//						mcHeight2MoveAbsolute.Execute		:=	TRUE;
//						mcHeight2MoveAbsolute.Position		:=	lrHeightReadyPosition;
//						IF mcHeight1MoveAbsolute.Done AND mcHeight2MoveAbsolute.Done THEN
//							mcHeight1MoveAbsolute.Execute	:=	FALSE;
//							mcHeight2MoveAbsolute.Execute	:=	FALSE;
//							eState							:=	E_Station.eReady;
//						END_IF	
//					ELSE
							eState							:=	E_Station.eReady;
//					END_IF	
			END_IF

	/////////////////////////////
		E_Station.eHoming:						// Stan bazowania 

			Homing();
			IF NOT bHoming THEN
			  	eState							:=	E_Station.ePreparingToReady;
			   	mcCartesianYManualMove.JogBackwards		:=FALSE;
				mcCartesianZManualMove.JogBackwards		:=FALSE;
				mcPreScrewerManualMove.JogBackwards		:=FALSE;
				mcCatcherManualMove.JogBackwards		:=FALSE;
				
				mcCartesianYManualMove.JogForward		:=FALSE;
				mcCartesianZManualMove.JogForward		:=FALSE;
				mcPreScrewerManualMove.JogForward		:=FALSE;
				mcCatcherManualMove.JogForward			:=FALSE;			
			END_IF		
			
	/////////////////////////////
		E_Station.eHomingDone:                  // Stan wykonania bazowania 
		
			bAdvancedHoming							:= FALSE;
			mcCartesianYManualMove.JogBackwards		:= FALSE;
			mcCartesianZManualMove.JogBackwards		:= FALSE;
			mcPreScrewerManualMove.JogBackwards		:= FALSE;
			mcCatcherManualMove.JogBackwards		:= FALSE;
			                                           
			mcCartesianYManualMove.JogForward		:= FALSE;
			mcCartesianZManualMove.JogForward		:= FALSE;
			mcPreScrewerManualMove.JogForward		:= FALSE;
			mcCatcherManualMove.JogForward			:= FALSE;
			                                           
			bHomingDone								:= TRUE;
			IF NOT bHoming THEN                 	
				eRunningState						:= E_CapPreScrewer.eReady;
			   	eState								:= E_Station.eReady;
			END_IF
			
	/////////////////////////////
		E_Station.ePreparingToReady:            // Stan przygotowywania do gotowosci (zawsze przed Ready)  

		//	IF tonDelayServoOn.Q(*bySafetyStateScrewer1.0 AND bySafetyStateScrewer2.0 AND bySafetyStateHightServo.0 *)THEN
				bCartesianYServoPower	:= nAxisYSafetyState.0;	// Przy pierwszym uruchomieniu Ustawienia Fabryczne robimy na wartość maksymalną
				bCartesianZServoPower	:= nAxisZSafetyState.0;	// Przy pierwszym uruchomieniu Ustawienia Fabryczne robimy na wartość maksymalną
				bPreScrewerPower		:= nAxisScrewSafetyState.0;
				bCatcherPower			:= nAxisCatcherSafetyState.0;
//				bStrawCatcherLiftEnable	:= TRUE;
		//	END_IF	
			
			IF mcCartesianYPower.Status AND mcCartesianZPower.Status AND mcPreScrewerPower.Status AND mcCatcherPower.Status  THEN 

				IF NOT bAxisYInPosition OR NOT bAxisZInPosition OR NOT bCartesianInReadyPos  THEN
					bHomingDone							:= FALSE;
					bHomingWithoutJiesang				:= fbStrawCatcherLift.bHomingDone;
				END_IF	
				 		
				eState									:=	E_Station.eReady;
			END_IF
			
         	IF bIgnoreError THEN
				eState										:=	E_Station.eReady;
			END_IF
	
	/////////////////////////////
		E_Station.ePreparingToDisable:          // Stan przygotowywania do nieaktywnosci (po wyłączeniu Enable) 
  
			bCartesianYServoPower	:= TRUE;	// Przy pierwszym uruchomieniu Ustawienia Fabryczne robimy na wartość maksymalną
			bCartesianZServoPower	:= TRUE;	// Przy pierwszym uruchomieniu Ustawienia Fabryczne robimy na wartość maksymalną
			bPreScrewerPower		:= TRUE;
			bCatcherPower			:= TRUE;
			
			eRunningState					:=	E_CapPreScrewer.eReady;		//Dodane
			PreparingToDisable();

         	IF bIgnoreError THEN
				eState:=E_Station.eDisabled;
			END_IF
			
	/////////////////////////////
		E_Station.eReady:						// Stan gotowosci 
		
		//Detekcja utraconej nasadki
			GVL_UVFF.ftVacuumSensor1(CLK := tonSuckedOk[1].Q);
			GVL_UVFF.ftVacuumSensor2(CLK := tonSuckedOk[2].Q);
			GVL_UVFF.ftVacuumSensor3(CLK := tonSuckedOk[3].Q);
			GVL_UVFF.ftVacuumSensor4(CLK := tonSuckedOk[4].Q);
		
				//Jeżeli utracimy nasadkę--> wyłącz ssawkę
			//bCapSucker[1]					R= GVL.ftVacuumSensor1.Q;
			//bCapSucker[2]					R= GVL.ftVacuumSensor2.Q;
			//bCapSucker[3]					R= GVL.ftVacuumSensor3.Q;
			//bCapSucker[4]					R= GVL.ftVacuumSensor4.Q;
			
			bEnableLift					:= FALSE;
		
		//Zdejmuję HomingDone gdy utracę bodaj jedną nasadkę lub Jiesang nie jest zbazowany
			//IF (*bAnyCapLost OR*) (NOT fbBottleCatch1Station.bHomingDone AND NOT bManualMovement) THEN
			//	bHomingDone					:= FALSE;
			//	bHomingWithoutJiesang		:= fbBottleCatch1Station.bHomingDone;
			//END_IF
		
			(*Skasowanie wszystkich komend*)
			IF rtResetCommands.Q THEN	
				ResetCommands();	
			END_IF
			
			IF bPreRun THEN
				eState						:= E_Station.eStarting;
			END_IF
			
			IF bRun AND NOT bCycleDone (*AND NOT bCycleNotDone*) AND bHomingDone THEN
				eState 						:= E_Station.eRunning; 
			END_IF
			IF bHoming THEN
				eState 						:= E_Station.eHoming; 
			END_IF
			
			IF NOT bRun THEN
				GVL_VIS.bCapSorterPreScrewerBottleCatcherCatch	:= FALSE;
				bPlaceDone										:= FALSE;
				bCycleDone 										:= FALSE;		
			END_IF
			
			IF bManualMovement THEN
				//Jeśli przejście w tryb ruchów manualnych przepisz wszystkie stany siłowników sterowanych przez moduł
				//aby zapobiec ewentualnym kolizjom po wejściu w tryb serwisowy
				//Ruchy manualne siłownika na wózku	
				bManualCapSucker1							:= bCapSucker[1];	
				bmanualCapSucker2							:= bCapSucker[2];	
				bManualCapSucker3							:= bCapSucker[3];	
				bManualCapSucker4							:= bCapSucker[4];	
				                          	    		                 
				bManualCapBlower1							:= bCapBlower1;	
				bManualCapBlower2							:= bCapBlower2;	
				bManualCapBlower3							:= bCapBlower3;	
				bManualCapBlower4							:= bCapBlower4;	
				                          		    	                 
				bManualCapCatcher1							:= bCapCatcher1;
				bManualCapCatcher2							:= bCapCatcher2;
				bManualCapCatcher3							:= bCapCatcher3;
				bManualCapCatcher4					    	:= bCapCatcher4;
				                                        	
				bManualStrawCatchersOpen					:= bStrawCatchersOpen;
				bManualStrawCatchersClose					:= bStrawCatchersClose;	                                            	
				                                        	
			    bManualStrawCatcherActuatorOut 				:= bStrawCatcherActuatorOut;
			    bManualStrawCatcherActuatorIn 				:= bStrawCatcherActuatorIn;
				
				bHomingWithoutJiesang						:= fbStrawCatcherLift.bHomingDone;
				
				eState 										:=	E_Station.eManualMovement; 

			END_IF
			
	/////////////////////////////
		E_Station.eStopping:					// Stan zatrzymywania 
			
			RunningCam();//RunningWithFlyingSaw();				//Running();
			
					IF bStopAllowed THEN
						eState 								:=	E_Station.eReady;
					END_IF

				
	/////////////////////////////
		E_Station.eStarting:                  	// Stan uruchamiania (po Ready)				
		
		IF 	eRunningState = E_CapPreScrewer.eReady THEN	//Jeżeli jesteśmy na poz. ready--> sprawdź i dojedź do pozycji home
				//Dojazd do poz top		                                                    	
			mcCartesianZMoveAbsolute.Execute						:= NOT bAxisZInTopPos;		
			mcCartesianZMoveAbsolute.Position						:= stParameters.lrTopZPosition;
			mcCartesianZMoveAbsolute.Acceleration					:= 500.0;
			mcCartesianZMoveAbsolute.Deceleration					:= 500.0;
			mcCartesianZMoveAbsolute.Velocity						:= 50;
			                                        				
			//najpierw os Z potem winda chwytakow   				
			mcCatcherMoveAbsolute.Execute							:= NOT bAxisStrawCatcherHomePos AND bAxisZInTopPos;		
			mcCatcherMoveAbsolute.Position							:= stParameters.lrCatcherCatchingPosition;
			mcCatcherMoveAbsolute.Acceleration						:= 300.0;
			mcCatcherMoveAbsolute.Deceleration						:= 300.0;
			mcCatcherMoveAbsolute.Velocity							:= 30;
			                                        				
			mcCartesianYMoveAbsolute.Execute						:= NOT bAxisYInHomePos AND bAxisZInTopPos;
			mcCartesianYMoveAbsolute.Position						:= stParameters.lrPickYPosition;
			mcCartesianYMoveAbsolute.Acceleration					:= 500.0;
			mcCartesianYMoveAbsolute.Deceleration					:= 500.0;
			mcCartesianYMoveAbsolute.Velocity						:= 50; 
			                                                    	
			IF bAxisZInTopPos THEN
				GVL_VIS.bCapSorterPreScrewerCatchStationHoming			:= NOT fbStrawCatcherLift.bHomingDone;
				GVL_VIS.bCapSorterPreScrewerCatcherStationHeightSet		:= NOT GVL_VIS.bCapSorterPreScrewerCatchStationHoming AND NOT bStrawCatcherLiftInHomePos;
				bEnableLift												:= TRUE;
			END_IF
    		
				IF 	bCartesianInTopPos AND bStrawCatcherLiftInHomePos THEN
					mcCartesianZMoveAbsolute.Execute              	:= FALSE;
					mcCatcherMoveAbsolute.Execute                 	:= FALSE;
					mcCartesianYMoveAbsolute.Execute              	:= FALSE;
					GVL_VIS.bCapSorterPreScrewerCatchStationHoming	:= FALSE;
					eState											:= E_Station.eRunning; 
				END_IF
		ELSE
			eState							:= E_Station.eRunning; 
			bEnableLift						:= TRUE;	
		END_IF	
					
			
	/////////////////////////////
		E_Station.eRunning:               		// Stan wykonywania cyklu (po Startingu), w tym stanie osobny
		
 			IF bRun THEN
				IF bSimulationEna THEN
					Simulation();
				ELSE	
					RunningCam();	//RunningWithFlyingSaw();				//Running();
				END_IF
				
				
			ELSIF NOT bPreRun THEN
				bBottleCatcherCatchTemp		:= FALSE;
				eState 				 		:= E_Station.eStopping;		
			END_IF
				
			
	/////////////////////////////	
		E_Station.eDone:
		
			IF bCycleDone THEN (*Cykl zakończony*)
				bBottleCatcherCatchTemp		:= FALSE;
			END_IF	
			
			IF NOT bPreRun  AND bStopAllowed THEN					(*Przerywanie cyklu*)
				bBottleCatcherCatchTemp		:= FALSE;
				eState 				 		:= E_Station.eStopping;	
			ELSIF NOT bRun THEN
				GVL_VIS.bCapSorterPreScrewerBottleCatcherCatch	:= FALSE;
				bPlaceDone										:= FALSE;
				bCycleDone 										:= FALSE;	
				eState 				 							:= E_Station.eRunning;	
			END_IF
		
		
		
	END_CASE

	
//IF (ABS(GVL_VIS.lrCapSorterPreScrewerCatcherStationHeightCV-stParameters.lrCatcherHightSV) > 2) AND
//	(eState = E_Station.eStarting OR eState = E_Station.ePreparingToReady) THEN
//			GVL_VIS.bCapSorterPreScrewerCatcherStationHeightSet 				:= TRUE;
//ELSIF ABS(GVL_VIS.lrCapSorterPreScrewerCatcherStationHeightCV-stParameters.lrCatcherHightSV) < 2 THEN
//			GVL_VIS.bCapSorterPreScrewerCatcherStationHeightSet 				:= FALSE;	
//END_IF
END_ACTION

ACTION ErrorHandling:
//CZYTANIE STATUSÓW
CartesianYAxisRef.ReadStatus();
CartesianZAxisRef.ReadStatus();
CatcherAxisRef.ReadStatus();
PreScrewerAxisRef.ReadStatus();
//Czasówki od siłowników
tonErrorStrawCatcherIn(IN:= bStrawCatcherActuatorIn AND NOT bStrawCatcherIn,PT:=T#1000MS);
tonErrorStrawCatcherOut(IN:= bStrawCatcherActuatorOut AND NOT bStrawCatcherOut,PT:=T#1000MS);



//**********************LISTA BŁĘDÓW******************************
bStateError	:= (eState=E_Station.eError) OR (eState=E_Station.eResetting) OR NOT bEstop OR bIgnoreError;

//PreparingToDisable i StateError ze względu na wciśnięcie EStopa podczas wyłączania i pojawienie się blędu
IF bEnable OR eState=E_Station.ePreparingToDisable THEN
	


	//Error 1 - BŁĄD SERWA POZIOMEGO X
	IF (CartesianYAxisRef.Status.Error OR mcCartesianYMoveAbsolute.Error) AND NOT arrFbAllarm[0].bActive THEN
		sAxisAlarm := CONCAT(UDINT_TO_STRING(CartesianYAxisRef.Status.ErrorID),F_AxErrMsg(CartesianYAxisRef.Status.ErrorID));
		arrFbAllarm[0].ipArguments.Clear().AddString(sAxisAlarm);		
		arrFbAllarm[0].Raise(nTimeStamp := 0);		
		udiErrorID							:=	1129;
		udiCartesianXServoErrorNr			:=	CartesianYAxisRef.Status.ErrorID;
		sErrorDescription					:=	'Błąd napędu poziomego Y. Błąd NC:';
		sErrorDescription2					:=	F_AX8xErrMsg(TO_UINT(udiCartesianXServoErrorNr));
	ELSIF NOT CartesianYAxisRef.Status.Error AND NOT mcCartesianYMoveAbsolute.Error AND eState = E_Station.eResetting AND arrFbAllarm[0].bActive THEN
			arrFbAllarm[0].Clear(nTimeStamp := 0, bResetConfirmation := FALSE);
	END_IF;
	
	//Error 2 - BŁĄD SERWA PIONOWEGO Z
	IF (CartesianZAxisRef.Status.Error OR mcCartesianZMoveAbsolute.Error) AND NOT arrFbAllarm[1].bActive THEN
		sAxisAlarm := CONCAT(UDINT_TO_STRING(CartesianZAxisRef.Status.ErrorID),F_AxErrMsg(CartesianZAxisRef.Status.ErrorID));
		arrFbAllarm[1].ipArguments.Clear().AddString(sAxisAlarm);		
		arrFbAllarm[1].Raise(nTimeStamp := 0);		
		udiErrorID							:=	1130;
		udiCartesianZServoErrorNr			:=	CartesianZAxisRef.Status.ErrorID;
		sErrorDescription					:=	'Błąd napędu podnoszenia Z. Błąd NC:';
		sErrorDescription2					:=	F_AX8xErrMsg(TO_UINT(udiCartesianZServoErrorNr));
	ELSIF NOT CartesianZAxisRef.Status.Error AND NOT mcCartesianZMoveAbsolute.Error AND eState = E_Station.eResetting AND arrFbAllarm[1].bActive THEN
			arrFbAllarm[1].Clear(nTimeStamp := 0, bResetConfirmation := FALSE);
	END_IF;
	
	//Error 3 - BŁĄD SERWA PIONOWEGO UCHWYTU SŁOMEK
	IF (CatcherAxisRef.Status.Error OR mcCatcherMoveAbsolute.Error) AND NOT arrFbAllarm[2].bActive THEN		
		sAxisAlarm := CONCAT(UDINT_TO_STRING(CatcherAxisRef.Status.ErrorID),F_AxErrMsg(CatcherAxisRef.Status.ErrorID));
		arrFbAllarm[2].ipArguments.Clear().AddString(sAxisAlarm);		
		arrFbAllarm[2].Raise(nTimeStamp := 0);		
		udiErrorID							:=	1131;
		udiCatcherServoErrorNr				:=	CatcherAxisRef.Status.ErrorID;
		sErrorDescription					:=	'Błąd napędu podnoszenia chwytaka słomek. Błąd NC:';
		sErrorDescription2					:=	F_AX8xErrMsg(TO_UINT(udiCatcherServoErrorNr));
	ELSIF NOT CatcherAxisRef.Status.Error AND NOT  mcCatcherMoveAbsolute.Error AND eState = E_Station.eResetting AND arrFbAllarm[2].bActive THEN
			arrFbAllarm[2].Clear(nTimeStamp := 0, bResetConfirmation := FALSE);
	END_IF;
	
	//Error 4 - BŁĄD SERWA OBROTOWEGO
	IF (PreScrewerAxisRef.Status.Error OR mcPreScrewerMoveAbsolute.Error OR bTestError) AND NOT arrFbAllarm[3].bActive THEN
		sAxisAlarm := CONCAT(UDINT_TO_STRING(PreScrewerAxisRef.Status.ErrorID),F_AxErrMsg(PreScrewerAxisRef.Status.ErrorID));
		arrFbAllarm[3].ipArguments.Clear().AddString(sAxisAlarm);		
		arrFbAllarm[3].Raise(nTimeStamp := 0);		
		udiErrorID							:=	1132;
		udiPreScrewerServoErrorNr			:=	PreScrewerAxisRef.Status.ErrorID;
		sErrorDescription					:=	'Błąd napędu zakręcania. Błąd NC:';
		sErrorDescription2					:=	F_AX8xErrMsg(TO_UINT(udiPreScrewerServoErrorNr));
	ELSIF NOT PreScrewerAxisRef.Status.Error AND NOT  mcPreScrewerMoveAbsolute.Error AND eState = E_Station.eResetting AND arrFbAllarm[3].bActive THEN
			arrFbAllarm[3].Clear(nTimeStamp := 0, bResetConfirmation := FALSE);
	END_IF;
	
	IF PreScrewerAxisRef.Status.Error THEN
		GVL_UVFF.diTest1	:= GVL_UVFF.diTest1 + 1;
	END_IF
	
	IF mcPreScrewerMoveAbsolute.Error THEN
		GVL_UVFF.diTest2	:= GVL_UVFF.diTest2 + 1;
	END_IF
	
	IF mcPreScrewerMoveRelative.Error THEN
		GVL_UVFF.diTesy3	:= GVL_UVFF.diTesy3 + 1;
	END_IF
	
	IF bTestError THEN
		GVL_UVFF.diTest4	:= GVL_UVFF.diTest4 + 1;
	END_IF	
	
	
	
	
	
	//Error 5A - BŁĄD PRZEKROCZENIE CZASU DZIAŁANIA SIŁOWNIKA CHWYTAKÓW SŁOMEK
	IF tonErrorStrawCatcherOut.Q AND NOT arrFbAllarm[4].bActive THEN
		arrFbAllarm[4].Raise(nTimeStamp := 0);	
		udiErrorID							:=	1133;
		udiPreScrewerServoErrorNr			:=	PreScrewerAxisRef.Status.ErrorID;
		sErrorDescription					:=	'Błąd siłownika chwytaków słomek | Zablokowany wysów';
		sErrorDescription2					:=	'';
	ELSIF NOT tonErrorStrawCatcherOut.Q AND eState = E_Station.eResetting AND arrFbAllarm[4].bActive THEN
			arrFbAllarm[4].Clear(nTimeStamp := 0, bResetConfirmation := FALSE);
	END_IF;
	
	//Error 5B - BŁĄD PRZEKROCZENIE CZASU DZIAŁANIA SIŁOWNIKA CHWYTAKÓW SŁOMEK
	IF tonErrorStrawCatcherIn.Q AND NOT arrFbAllarm[5].bActive THEN
		arrFbAllarm[5].Raise(nTimeStamp := 0);	
		udiErrorID							:=	1134;
		udiPreScrewerServoErrorNr			:=	PreScrewerAxisRef.Status.ErrorID;
		sErrorDescription					:=	'Błąd siłownika chwytaków słomek | Zablokowane cofnięcie';
		sErrorDescription2					:=	'';
	ELSIF NOT tonErrorStrawCatcherIn.Q AND eState = E_Station.eResetting AND arrFbAllarm[5].bActive THEN
			arrFbAllarm[5].Clear(nTimeStamp := 0, bResetConfirmation := FALSE);
	END_IF;
	
	//Error 6 - Blad podnosnika Jiecang - brak zasilania lub zablokowany mechanicznie
	IF fbStrawCatcherLift.bError AND fbStrawCatcherLift.nErrorNr = 1 AND NOT arrFbAllarm[6].bActive THEN
		arrFbAllarm[6].Raise(nTimeStamp := 0);	
    	udiErrorID				:= 1135;
    	sErrorDescription		:= 'Błąd podnosnika lub brak zasilania';
    	sErrorDescription2		:= ' ';
	ELSIF NOT fbStrawCatcherLift.bError AND eState = E_Station.eResetting AND arrFbAllarm[6].bActive THEN
			arrFbAllarm[6].Clear(nTimeStamp := 0, bResetConfirmation := FALSE);
	END_IF;
		

	//Error 6 - Blad podnosnika Jiecang - prak zasilania lub zablokowany mechanicznie
	IF fbStrawCatcherLift.bError AND fbStrawCatcherLift.nErrorNr = 2 AND NOT arrFbAllarm[7].bActive THEN
		arrFbAllarm[7].Raise(nTimeStamp := 0);
    	udiErrorID				:= 1136;
    	sErrorDescription		:= 'Błąd podnosnika  - wartość zadana jest większa od wartości maksymalnej';
    	sErrorDescription2		:= ' ';
	ELSIF NOT fbStrawCatcherLift.bError AND eState = E_Station.eResetting AND arrFbAllarm[7].bActive THEN
			arrFbAllarm[7].Clear(nTimeStamp := 0, bResetConfirmation := FALSE);
	END_IF;
	
	
	//Error 6 - Blad podnosnika Jiecang - prak zasilania lub zablokowany mechanicznie
	IF  fbStrawCatcherLift.bError AND fbStrawCatcherLift.nErrorNr = 3 AND NOT arrFbAllarm[8].bActive THEN
		arrFbAllarm[8].Raise(nTimeStamp := 0);
    	udiErrorID				:= 1137;
    	sErrorDescription		:= 'Błąd podnosnika - wartość zadana jest mniejsza od wartości minimalnej';
    	sErrorDescription2		:= ' ';
	ELSIF NOT fbStrawCatcherLift.bError AND eState = E_Station.eResetting AND arrFbAllarm[8].bActive THEN
			arrFbAllarm[8].Clear(nTimeStamp := 0, bResetConfirmation := FALSE);
	END_IF;
	
		//Error 11 - Blad Kolizja	
	IF  rtCollisionError.Q AND NOT arrFbAllarm[13].bActive THEN
		arrFbAllarm[13].Raise(nTimeStamp := 0);
    	udiErrorID				:= 1142;
    	sErrorDescription		:= 'Kolizja kartezjana z transporterem nakrętek | Zbazuj stacje wkładania nakrętek';
    	sErrorDescription2		:= '';
	ELSIF NOT  rtCollisionError.Q AND eState = E_Station.eResetting AND arrFbAllarm[13].bActive THEN
			arrFbAllarm[13].Clear(nTimeStamp := 0, bResetConfirmation := FALSE);
	END_IF;

		//Przekroczona ilość prób pobrania nasadki, mówer1, słot1
	IF diMover1VacuumRetry[1] >= 3  AND NOT arrFbAllarm[14].bActive THEN
		arrFbAllarm[14].Raise(nTimeStamp := 0);
    	udiErrorID				:= 1143;
    	sErrorDescription		:= 'Przekroczona ilość prób pobrania nasadki, wózek1, slot1';
    	sErrorDescription2		:= '';
	ELSIF diMover1VacuumRetry[1] < 3 AND eState = E_Station.eResetting AND arrFbAllarm[14].bActive THEN
			arrFbAllarm[14].Clear(nTimeStamp := 0, bResetConfirmation := FALSE);
	END_IF;
	
	IF diMover1VacuumRetry[2] >= 3  AND NOT arrFbAllarm[15].bActive THEN
		arrFbAllarm[15].Raise(nTimeStamp := 0);
    	udiErrorID				:= 1144;
    	sErrorDescription		:= 'Przekroczona ilość prób pobrania nasadki, wózek1, slot2';
    	sErrorDescription2		:= '';
	ELSIF diMover1VacuumRetry[2] < 3 AND eState = E_Station.eResetting AND arrFbAllarm[15].bActive THEN
			arrFbAllarm[15].Clear(nTimeStamp := 0, bResetConfirmation := FALSE);
	END_IF;

	IF diMover1VacuumRetry[3] >= 3  AND NOT arrFbAllarm[16].bActive THEN
		arrFbAllarm[16].Raise(nTimeStamp := 0);
    	udiErrorID				:= 1145;
    	sErrorDescription		:= 'Przekroczona ilość prób pobrania nasadki, wózek1, slot3';
    	sErrorDescription2		:= '';
	ELSIF diMover1VacuumRetry[3] < 3 AND eState = E_Station.eResetting AND arrFbAllarm[16].bActive THEN
			arrFbAllarm[16].Clear(nTimeStamp := 0, bResetConfirmation := FALSE);
	END_IF;
	
	IF diMover1VacuumRetry[4] >= 3  AND NOT arrFbAllarm[17].bActive THEN
		arrFbAllarm[17].Raise(nTimeStamp := 0);
    	udiErrorID				:= 1146;
    	sErrorDescription		:= 'Przekroczona ilość prób pobrania nasadki, wózek1, slot4';
    	sErrorDescription2		:= '';
	ELSIF diMover1VacuumRetry[4] < 3 AND eState = E_Station.eResetting AND arrFbAllarm[17].bActive THEN
			arrFbAllarm[17].Clear(nTimeStamp := 0, bResetConfirmation := FALSE);
	END_IF;
	
			//Przekroczona ilość prób pobrania nasadki, mówer2, słot1
	IF diMover2VacuumRetry[1] >= 3  AND NOT arrFbAllarm[18].bActive THEN
		arrFbAllarm[18].Raise(nTimeStamp := 0);
    	udiErrorID				:= 1147;
    	sErrorDescription		:= 'Przekroczona ilość prób pobrania nasadki, wózek2, slot1';
    	sErrorDescription2		:= '';
	ELSIF diMover2VacuumRetry[1] < 3 AND eState = E_Station.eResetting AND arrFbAllarm[18].bActive THEN
			arrFbAllarm[18].Clear(nTimeStamp := 0, bResetConfirmation := FALSE);
	END_IF;
	
	IF diMover2VacuumRetry[2] >= 3  AND NOT arrFbAllarm[19].bActive THEN
		arrFbAllarm[19].Raise(nTimeStamp := 0);
    	udiErrorID				:= 1148;
    	sErrorDescription		:= 'Przekroczona ilość prób pobrania nasadki, wózek2, slot2';
    	sErrorDescription2		:= '';
	ELSIF diMover2VacuumRetry[2] < 3 AND eState = E_Station.eResetting AND arrFbAllarm[19].bActive THEN
			arrFbAllarm[19].Clear(nTimeStamp := 0, bResetConfirmation := FALSE);
	END_IF;

	IF diMover2VacuumRetry[3] >= 3  AND NOT arrFbAllarm[20].bActive THEN
		arrFbAllarm[20].Raise(nTimeStamp := 0);
    	udiErrorID				:= 1149;
    	sErrorDescription		:= 'Przekroczona ilość prób pobrania nasadki, wózek2, slot3';
    	sErrorDescription2		:= '';
	ELSIF diMover2VacuumRetry[3] < 3 AND eState = E_Station.eResetting AND arrFbAllarm[20].bActive THEN
			arrFbAllarm[20].Clear(nTimeStamp := 0, bResetConfirmation := FALSE);
	END_IF;
	
	IF diMover2VacuumRetry[4] >= 3  AND NOT arrFbAllarm[21].bActive THEN
		arrFbAllarm[21].Raise(nTimeStamp := 0);
    	udiErrorID				:= 1150;
    	sErrorDescription		:= 'Przekroczona ilość prób pobrania nasadki, wózek2, slot4';
    	sErrorDescription2		:= '';
	ELSIF diMover2VacuumRetry[4] < 3 AND eState = E_Station.eResetting AND arrFbAllarm[21].bActive THEN
			arrFbAllarm[21].Clear(nTimeStamp := 0, bResetConfirmation := FALSE);
	END_IF;

	IF NOT arrFbAllarm[22].bActive AND (fbVirtualAxis.bErrorFB  OR fbVirtualAxis.bError) THEN	
		sAxisAlarm := CONCAT(UDINT_TO_STRING(fbVirtualAxis.nErrorId),F_AxErrMsg(fbVirtualAxis.nErrorId));
		arrFbAllarm[22].ipArguments.Clear().AddString(sAxisAlarm);		
		arrFbAllarm[22].Raise(nTimeStamp := 0);	
		udiErrorID							:=	1151;
		sErrorDescription					:=	'Błąd wirtualnej osi:';
		sErrorDescription2					:=	F_AX8xErrMsg(TO_UINT(fbVirtualAxis.nErrorId));
	ELSIF NOT fbVirtualAxis.bError AND NOT  fbVirtualAxis.bErrorFB AND eState = E_Station.eResetting AND arrFbAllarm[22].bActive THEN
			arrFbAllarm[22].Clear(nTimeStamp := 0, bResetConfirmation := FALSE);
	END_IF;
	
	IF (fbVirtualAxis.pSetPos.Error OR fbVirtualAxis.pSetPos.CommandAborted) AND NOT arrFbAllarm[23].bActive THEN
		arrFbAllarm[23].ipArguments.Clear().AddUDInt(fbVirtualAxis.pSetPos.ErrorID);		
		arrFbAllarm[23].Raise(nTimeStamp := 0);		
    	udiErrorID							:= 1152;
    	udiErrorID							:= udiErrorID + iStationIndex;
    	sErrorDescription					:= CONCAT('Błąd wirtualnej osi', UDINT_TO_STRING(fbVirtualAxis.pSetPos.ErrorID));
    	sErrorDescription2					:= ' ';	
	ELSIF NOT fbVirtualAxis.pSetPos.Error AND eState = E_Station.eResetting AND arrFbAllarm[23].bActive THEN
			arrFbAllarm[23].Clear(nTimeStamp := 0, bResetConfirmation := FALSE);
	END_IF;
	
	IF fbCamTableSelectAxisZ.Error AND NOT arrFbAllarm[24].bActive THEN
		arrFbAllarm[24].ipArguments.Clear().AddUDInt(fbCamTableSelectAxisZ.ErrorID);		
		arrFbAllarm[24].Raise(nTimeStamp := 0);		
    	udiErrorID							:= 1154;
    	udiErrorID							:= udiErrorID + iStationIndex;
    	sErrorDescription					:= CONCAT('Błąd generowania krzywki osi Z, MC_CamTableSelect.ErrorID:', UDINT_TO_STRING(fbCamTableSelectAxisZ.ErrorID));
    	sErrorDescription2					:= ' ';	
	ELSIF NOT fbCamTableSelectAxisZ.Error AND eState = E_Station.eResetting AND arrFbAllarm[24].bActive THEN
			arrFbAllarm[24].Clear(nTimeStamp := 0, bResetConfirmation := FALSE);
	END_IF;
	
	IF fbCamTableSelectCatcher.Error AND NOT arrFbAllarm[25].bActive THEN
		arrFbAllarm[25].ipArguments.Clear().AddUDInt(fbCamTableSelectCatcher.ErrorID);		
		arrFbAllarm[25].Raise(nTimeStamp := 0);		
    	udiErrorID							:= 1155;
    	udiErrorID							:= udiErrorID + iStationIndex;
    	sErrorDescription					:= CONCAT('Błąd generowania krzywki osi prowadzenia słomki, MC_CamTableSelect.ErrorID:', UDINT_TO_STRING(fbCamTableSelectCatcher.ErrorID));
    	sErrorDescription2					:= ' ';	
	ELSIF NOT fbCamTableSelectCatcher.Error AND eState = E_Station.eResetting AND arrFbAllarm[25].bActive THEN
			arrFbAllarm[25].Clear(nTimeStamp := 0, bResetConfirmation := FALSE);
	END_IF;
	
	IF fbCamInAxisZ.Error AND NOT arrFbAllarm[26].bActive THEN
		arrFbAllarm[26].ipArguments.Clear().AddUDInt(fbCamInAxisZ.ErrorID);		
		arrFbAllarm[26].Raise(nTimeStamp := 0);		
    	udiErrorID							:= 1156;
    	udiErrorID							:= udiErrorID + iStationIndex;
    	sErrorDescription					:= CONCAT('Błąd synchronizacji osi Z, MC_CamIn.ErrorID: ', UDINT_TO_STRING(fbCamInAxisZ.ErrorID));
    	sErrorDescription2					:= ' ';	
	ELSIF NOT fbCamInAxisZ.Error AND eState = E_Station.eResetting AND arrFbAllarm[26].bActive THEN
			arrFbAllarm[26].Clear(nTimeStamp := 0, bResetConfirmation := FALSE);
	END_IF;
	
	IF fbCamInAxisCatcher.Error AND NOT arrFbAllarm[27].bActive THEN
		arrFbAllarm[27].ipArguments.Clear().AddUDInt(fbCamInAxisCatcher.ErrorID);		
		arrFbAllarm[27].Raise(nTimeStamp := 0);		
    	udiErrorID							:= 1157;
    	udiErrorID							:= udiErrorID + iStationIndex;
    	sErrorDescription					:= CONCAT('Błąd synchronizacji osi prowadzenia słomki, MC_CamIn.ErrorID:', UDINT_TO_STRING(fbCamInAxisCatcher.ErrorID));
    	sErrorDescription2					:= ' ';	
	ELSIF NOT fbCamInAxisCatcher.Error AND eState = E_Station.eResetting AND arrFbAllarm[27].bActive THEN
			arrFbAllarm[27].Clear(nTimeStamp := 0, bResetConfirmation := FALSE);
	END_IF;
	
	IF fbCamOutAxisZ.Error AND NOT arrFbAllarm[28].bActive THEN
		arrFbAllarm[28].ipArguments.Clear().AddUDInt(fbCamOutAxisZ.ErrorID);		
		arrFbAllarm[28].Raise(nTimeStamp := 0);		
    	udiErrorID							:= 1158;
    	udiErrorID							:= udiErrorID + iStationIndex;
    	sErrorDescription					:= CONCAT('Błąd rozsynchronizacji osi Z, MCCamOut.ErrorID:', UDINT_TO_STRING(fbCamOutAxisZ.ErrorID));
    	sErrorDescription2					:= ' ';	
	ELSIF NOT fbCamOutAxisZ.Error AND eState = E_Station.eResetting AND arrFbAllarm[28].bActive THEN
			arrFbAllarm[28].Clear(nTimeStamp := 0, bResetConfirmation := FALSE);
	END_IF;
	
	IF fbCamOutAxisCatcher.Error AND NOT arrFbAllarm[29].bActive THEN
		arrFbAllarm[29].ipArguments.Clear().AddUDInt(fbCamOutAxisCatcher.ErrorID);		
		arrFbAllarm[29].Raise(nTimeStamp := 0);		
    	udiErrorID							:= 1159;
    	udiErrorID							:= udiErrorID + iStationIndex;
    	sErrorDescription					:= CONCAT('Błąd rozsynchronizacji osi prowadzenia słomki, MCCamOut.ErrorID:', UDINT_TO_STRING(fbCamOutAxisCatcher.ErrorID));
    	sErrorDescription2					:= ' ';	
	ELSIF NOT fbCamOutAxisCatcher.Error AND eState = E_Station.eResetting AND arrFbAllarm[29].bActive THEN
			arrFbAllarm[29].Clear(nTimeStamp := 0, bResetConfirmation := FALSE);
	END_IF;
	
	FOR i:= 0 TO 23 DO
		bError S= arrFbAllarm[i].bActive;
	END_FOR
	
ELSE
	bError := FALSE;
END_IF


//******************PRZEJŚCIE DO eERROR*****************************


IF bError AND NOT bStateError THEN
	IF eLastState = E_Station.eRunning THEN
		bCycleNotDone 			:= FALSE;
	END_IF
	eState := E_Station.eError;
	ResetCommands();
END_IF

//****************WYŚWIETLANIE STATUSU BLEDU***********************

(*Wyświetlanie błedu na wyjściu*)
bError;

(*Przepisywanie nazwy stacji*)
sErrorStationName := wsLiteral_TO_UTF8(wsStationName);

(*Kasowanie casów resettingu*)
//IF  udiErrorID-iStationIndex <>3 THEN
//	iErrorResseting3	:=	0;
//END_IF
END_ACTION

ACTION FBs:
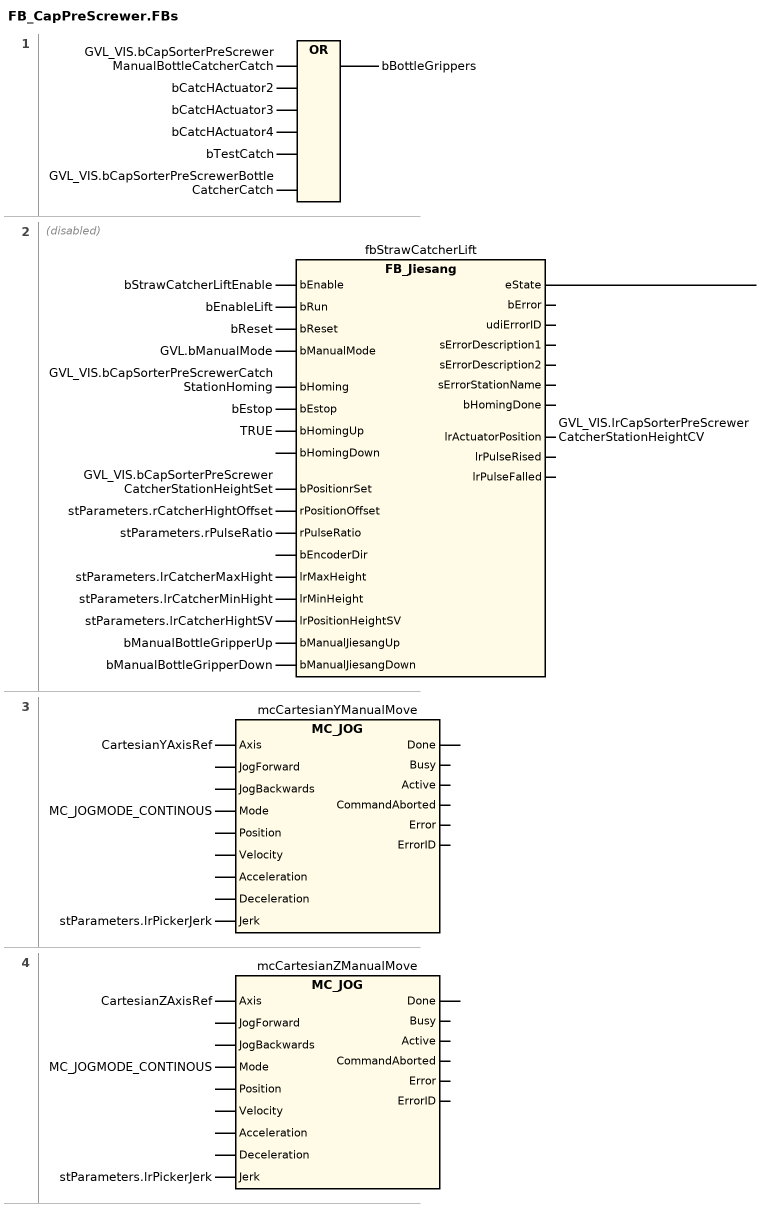
// NETWORK 1
bBottleGrippers := GVL_VIS.bCapSorterPreScrewerManualBottleCatcherCatch OR bCatcHActuator2 OR bCatcHActuator3 OR bCatcHActuator4 OR bTestCatch OR GVL_VIS.bCapSorterPreScrewerBottleCatcherCatch;

// NETWORK 2 (disabled)
// fbStrawCatcherLift(
//     bEnable := bStrawCatcherLiftEnable,
//     bRun := bEnableLift,
//     bReset := bReset,
//     bManualMode := GVL.bManualMode,
//     bHoming := GVL_VIS.bCapSorterPreScrewerCatchStationHoming,
//     bEstop := bEstop,
//     bHomingUp := TRUE,
//     bPositionrSet := GVL_VIS.bCapSorterPreScrewerCatcherStationHeightSet,
//     rPositionOffset := stParameters.rCatcherHightOffset,
//     rPulseRatio := stParameters.rPulseRatio,
//     lrMaxHeight := stParameters.lrCatcherMaxHight,
//     lrMinHeight := stParameters.lrCatcherMinHight,
//     lrPositionHeightSV := stParameters.lrCatcherHightSV,
//     bManualJiesangUp := bManualBottleGripperUp,
//     bManualJiesangDown := bManualBottleGripperDown,
//     lrActuatorPosition => GVL_VIS.lrCapSorterPreScrewerCatcherStationHeightCV); // FB_Jiesang

// NETWORK 3
mcCartesianYManualMove(
    Axis := CartesianYAxisRef,
    Mode := MC_JOGMODE_CONTINOUS,
    Jerk := stParameters.lrPickerJerk); // MC_JOG

// NETWORK 4
mcCartesianZManualMove(
    Axis := CartesianZAxisRef,
    Mode := MC_JOGMODE_CONTINOUS,
    Jerk := stParameters.lrPickerJerk); // MC_JOG

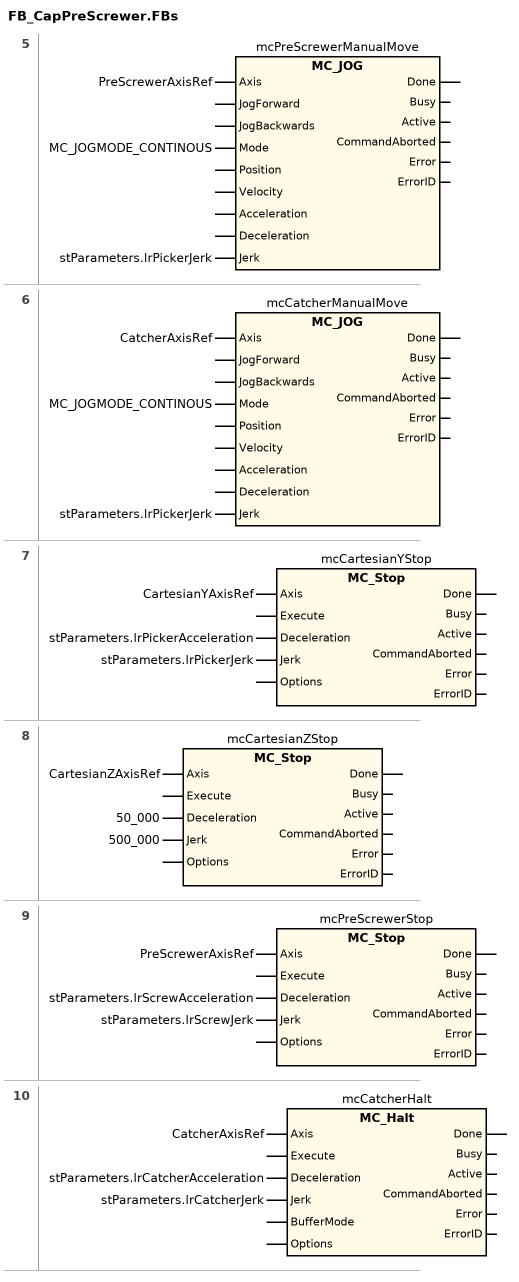
// NETWORK 5
mcPreScrewerManualMove(
    Axis := PreScrewerAxisRef,
    Mode := MC_JOGMODE_CONTINOUS,
    Jerk := stParameters.lrPickerJerk); // MC_JOG

// NETWORK 6
mcCatcherManualMove(Axis := CatcherAxisRef, Mode := MC_JOGMODE_CONTINOUS, Jerk := stParameters.lrPickerJerk); // MC_JOG

// NETWORK 7
mcCartesianYStop(
    Axis := CartesianYAxisRef,
    Deceleration := stParameters.lrPickerAcceleration,
    Jerk := stParameters.lrPickerJerk); // MC_Stop

// NETWORK 8
mcCartesianZStop(Axis := CartesianZAxisRef, Deceleration := 50_000, Jerk := 500_000); // MC_Stop

// NETWORK 9
mcPreScrewerStop(
    Axis := PreScrewerAxisRef,
    Deceleration := stParameters.lrScrewAcceleration,
    Jerk := stParameters.lrScrewJerk); // MC_Stop

// NETWORK 10
mcCatcherHalt(
    Axis := CatcherAxisRef,
    Deceleration := stParameters.lrCatcherAcceleration,
    Jerk := stParameters.lrCatcherJerk); // MC_Halt

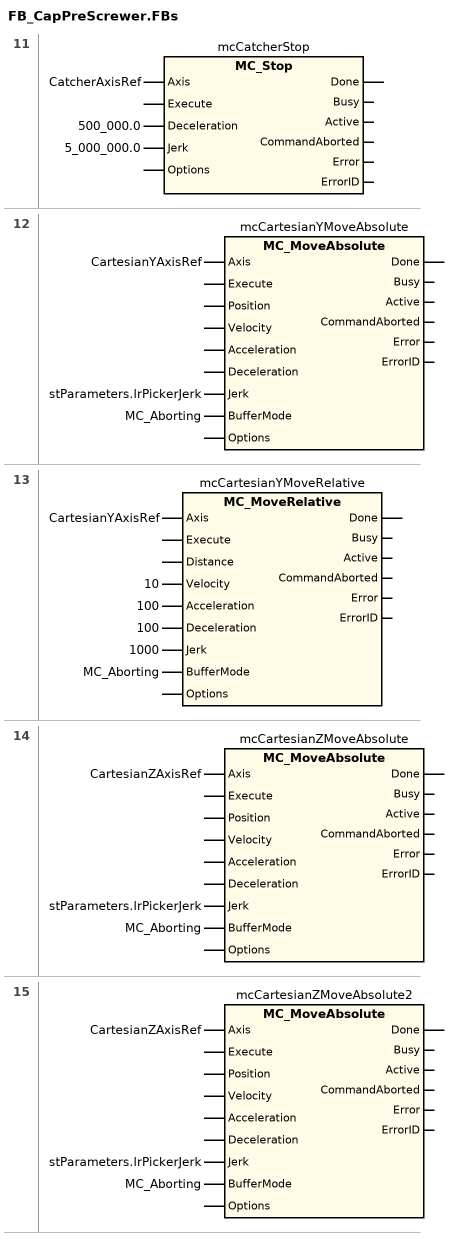
// NETWORK 11
mcCatcherStop(Axis := CatcherAxisRef, Deceleration := 500_000.0, Jerk := 5_000_000.0); // MC_Stop

// NETWORK 12
mcCartesianYMoveAbsolute(
    Axis := CartesianYAxisRef,
    Jerk := stParameters.lrPickerJerk,
    BufferMode := MC_Aborting); // MC_MoveAbsolute

// NETWORK 13
mcCartesianYMoveRelative(
    Axis := CartesianYAxisRef,
    Velocity := 10,
    Acceleration := 100,
    Deceleration := 100,
    Jerk := 1000,
    BufferMode := MC_Aborting); // MC_MoveRelative

// NETWORK 14
mcCartesianZMoveAbsolute(
    Axis := CartesianZAxisRef,
    Jerk := stParameters.lrPickerJerk,
    BufferMode := MC_Aborting); // MC_MoveAbsolute

// NETWORK 15
mcCartesianZMoveAbsolute2(
    Axis := CartesianZAxisRef,
    Jerk := stParameters.lrPickerJerk,
    BufferMode := MC_Aborting); // MC_MoveAbsolute

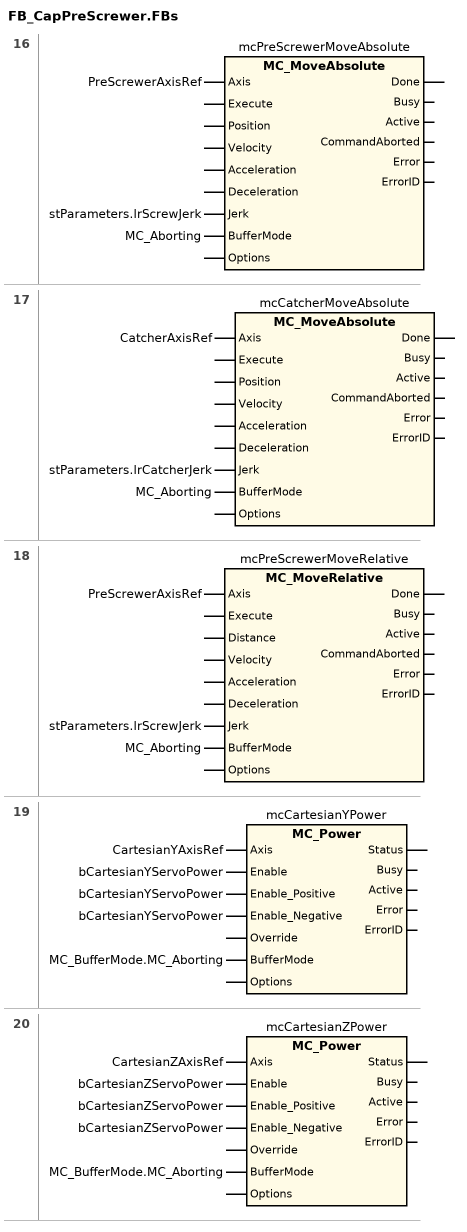
// NETWORK 16
mcPreScrewerMoveAbsolute(
    Axis := PreScrewerAxisRef,
    Jerk := stParameters.lrScrewJerk,
    BufferMode := MC_Aborting); // MC_MoveAbsolute

// NETWORK 17
mcCatcherMoveAbsolute(Axis := CatcherAxisRef, Jerk := stParameters.lrCatcherJerk, BufferMode := MC_Aborting); // MC_MoveAbsolute

// NETWORK 18
mcPreScrewerMoveRelative(
    Axis := PreScrewerAxisRef,
    Jerk := stParameters.lrScrewJerk,
    BufferMode := MC_Aborting); // MC_MoveRelative

// NETWORK 19
mcCartesianYPower(
    Axis := CartesianYAxisRef,
    Enable := bCartesianYServoPower,
    Enable_Positive := bCartesianYServoPower,
    Enable_Negative := bCartesianYServoPower,
    BufferMode := MC_BufferMode.MC_Aborting); // MC_Power

// NETWORK 20
mcCartesianZPower(
    Axis := CartesianZAxisRef,
    Enable := bCartesianZServoPower,
    Enable_Positive := bCartesianZServoPower,
    Enable_Negative := bCartesianZServoPower,
    BufferMode := MC_BufferMode.MC_Aborting); // MC_Power

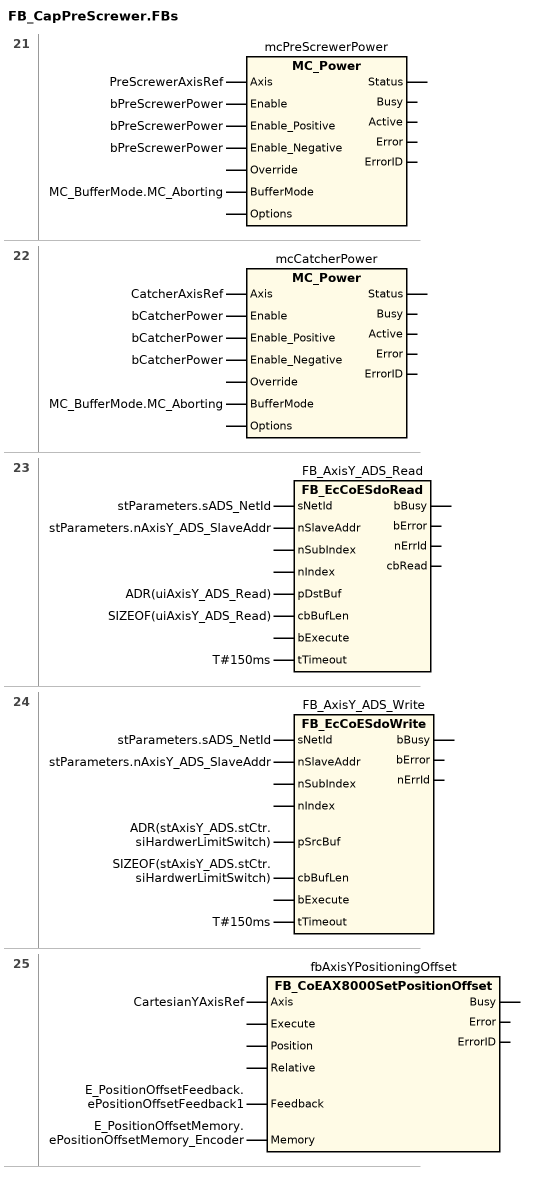
// NETWORK 21
mcPreScrewerPower(
    Axis := PreScrewerAxisRef,
    Enable := bPreScrewerPower,
    Enable_Positive := bPreScrewerPower,
    Enable_Negative := bPreScrewerPower,
    BufferMode := MC_BufferMode.MC_Aborting); // MC_Power

// NETWORK 22
mcCatcherPower(
    Axis := CatcherAxisRef,
    Enable := bCatcherPower,
    Enable_Positive := bCatcherPower,
    Enable_Negative := bCatcherPower,
    BufferMode := MC_BufferMode.MC_Aborting); // MC_Power

// NETWORK 23
FB_AxisY_ADS_Read(
    sNetId := stParameters.sADS_NetId,
    nSlaveAddr := stParameters.nAxisY_ADS_SlaveAddr,
    pDstBuf := ADR(uiAxisY_ADS_Read),
    cbBufLen := SIZEOF(uiAxisY_ADS_Read),
    tTimeout := T#150ms); // FB_EcCoESdoRead

// NETWORK 24
FB_AxisY_ADS_Write(
    sNetId := stParameters.sADS_NetId,
    nSlaveAddr := stParameters.nAxisY_ADS_SlaveAddr,
    pSrcBuf := ADR(stAxisY_ADS.stCtr.siHardwerLimitSwitch),
    cbBufLen := SIZEOF(stAxisY_ADS.stCtr.siHardwerLimitSwitch),
    tTimeout := T#150ms); // FB_EcCoESdoWrite

// NETWORK 25
fbAxisYPositioningOffset(
    Axis := CartesianYAxisRef,
    Feedback := E_PositionOffsetFeedback.ePositionOffsetFeedback1,
    Memory := E_PositionOffsetMemory.ePositionOffsetMemory_Encoder); // FB_CoEAX8000SetPositionOffset

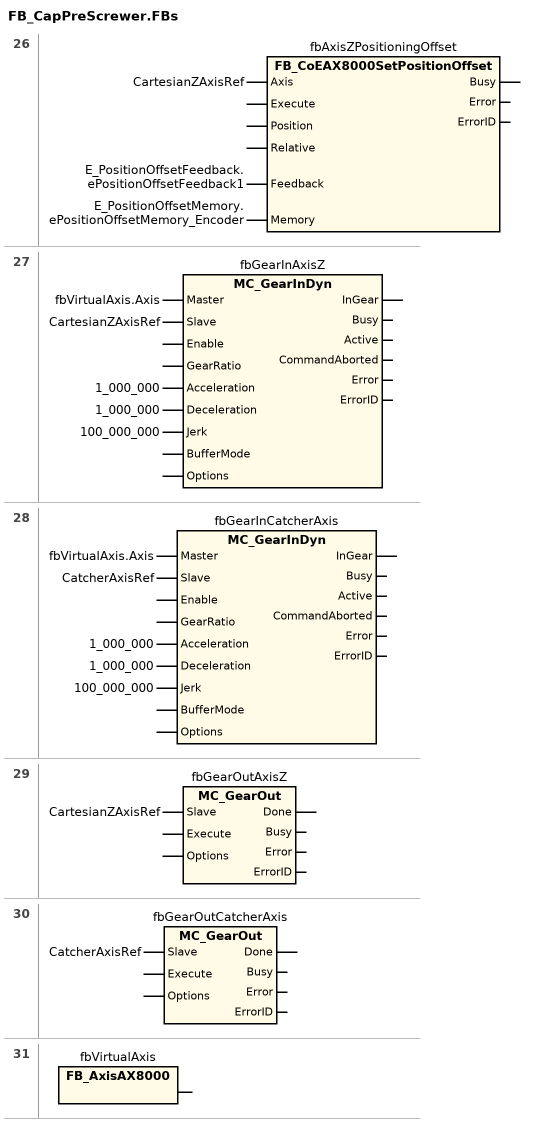
// NETWORK 26
fbAxisZPositioningOffset(
    Axis := CartesianZAxisRef,
    Feedback := E_PositionOffsetFeedback.ePositionOffsetFeedback1,
    Memory := E_PositionOffsetMemory.ePositionOffsetMemory_Encoder); // FB_CoEAX8000SetPositionOffset

// NETWORK 27
fbGearInAxisZ(
    Master := fbVirtualAxis.Axis,
    Slave := CartesianZAxisRef,
    Acceleration := 1_000_000,
    Deceleration := 1_000_000,
    Jerk := 100_000_000); // MC_GearInDyn

// NETWORK 28
fbGearInCatcherAxis(
    Master := fbVirtualAxis.Axis,
    Slave := CatcherAxisRef,
    Acceleration := 1_000_000,
    Deceleration := 1_000_000,
    Jerk := 100_000_000); // MC_GearInDyn

// NETWORK 29
fbGearOutAxisZ(Slave := CartesianZAxisRef); // MC_GearOut

// NETWORK 30
fbGearOutCatcherAxis(Slave := CatcherAxisRef); // MC_GearOut

// NETWORK 31
fbVirtualAxis(); // FB_AxisAX8000

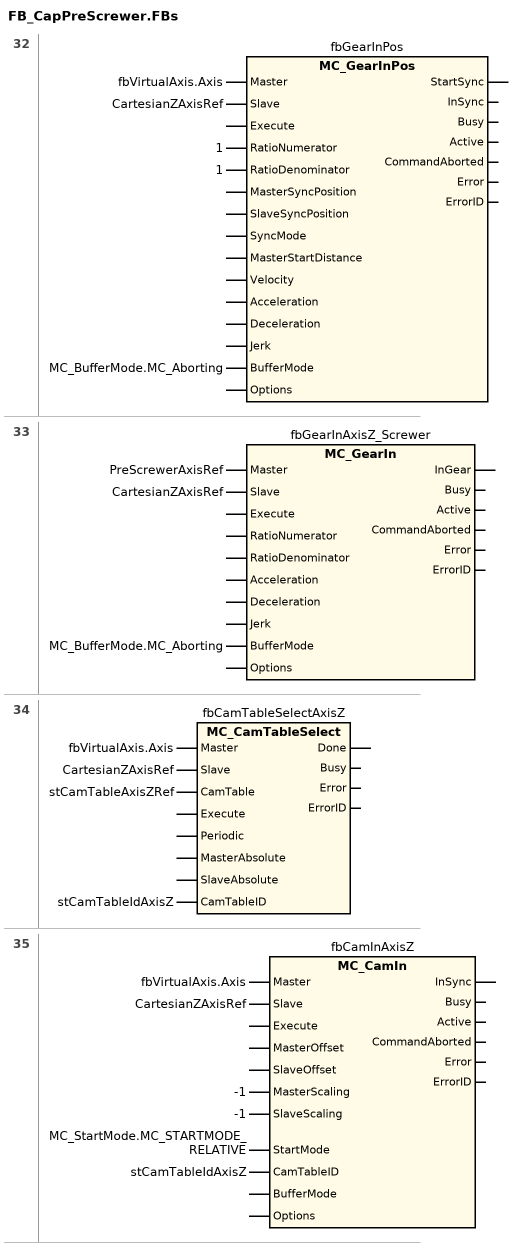
// NETWORK 32
fbGearInPos(
    Master := fbVirtualAxis.Axis,
    Slave := CartesianZAxisRef,
    RatioNumerator := 1,
    RatioDenominator := 1,
    BufferMode := MC_BufferMode.MC_Aborting); // MC_GearInPos

// NETWORK 33
fbGearInAxisZ_Screwer(
    Master := PreScrewerAxisRef,
    Slave := CartesianZAxisRef,
    BufferMode := MC_BufferMode.MC_Aborting); // MC_GearIn

// NETWORK 34
fbCamTableSelectAxisZ(
    Master := fbVirtualAxis.Axis,
    Slave := CartesianZAxisRef,
    CamTable := stCamTableAxisZRef,
    CamTableID := stCamTableIdAxisZ); // MC_CamTableSelect

// NETWORK 35
fbCamInAxisZ(
    Master := fbVirtualAxis.Axis,
    Slave := CartesianZAxisRef,
    MasterScaling := -1,
    SlaveScaling := -1,
    StartMode := MC_StartMode.MC_STARTMODE_RELATIVE,
    CamTableID := stCamTableIdAxisZ); // MC_CamIn

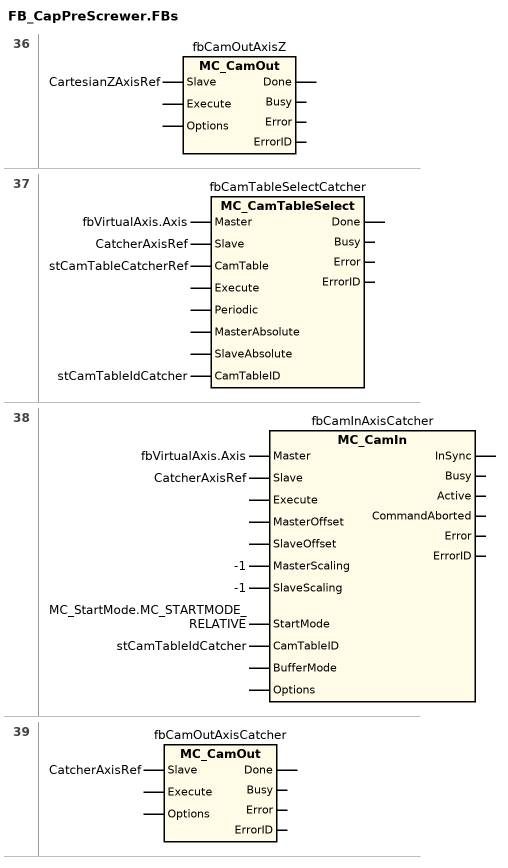
// NETWORK 36
fbCamOutAxisZ(Slave := CartesianZAxisRef); // MC_CamOut

// NETWORK 37
fbCamTableSelectCatcher(
    Master := fbVirtualAxis.Axis,
    Slave := CatcherAxisRef,
    CamTable := stCamTableCatcherRef,
    CamTableID := stCamTableIdCatcher); // MC_CamTableSelect

// NETWORK 38
fbCamInAxisCatcher(
    Master := fbVirtualAxis.Axis,
    Slave := CatcherAxisRef,
    MasterScaling := -1,
    SlaveScaling := -1,
    StartMode := MC_StartMode.MC_STARTMODE_RELATIVE,
    CamTableID := stCamTableIdCatcher); // MC_CamIn

// NETWORK 39
fbCamOutAxisCatcher(Slave := CatcherAxisRef); // MC_CamOut
END_ACTION

ACTION Homing:
tonAxisYLagDetction(PT := T#250MS);

IF mcCartesianZPower.Status AND mcPreScrewerPower.Status AND mcCatcherPower.Status THEN
		
	IF bHoming THEN // Bazowanie - podjazd do góry i ustawienie obrotu
		IF NOT bAdvancedHoming THEN
			CASE iHomingCase OF
			
				0:
					mcCartesianYPower.Override			:=	100;			
					mcCartesianZPower.Override			:=	100;			
					mcPreScrewerPower.Override			:=	100;			
					mcCatcherPower.Override				:=	100;	
					                                    
					bCartesianYServoPower				:= TRUE;
					bCartesianZServoPower				:= TRUE;
					bPreScrewerPower					:= TRUE;
					bCatcherPower						:= TRUE;	
					                                    
					mcCartesianYManualMove.JogBackwards	:=FALSE;
					mcCartesianZManualMove.JogBackwards	:=FALSE;
					mcPreScrewerManualMove.JogBackwards	:=FALSE;
					mcCatcherManualMove.JogBackwards	:=FALSE;
					                                    
					mcCartesianYManualMove.JogForward	:=FALSE;
					mcCartesianZManualMove.JogForward	:=FALSE;
					mcPreScrewerManualMove.JogForward	:=FALSE;
					mcCatcherManualMove.JogForward		:=FALSE;
					bCycleNotDone						:= FALSE;				
					
					IF bAnyCapPresence THEN
						iHomingCase						:= iHomingCase	+	100;
					ELSE
						iHomingCase						:= iHomingCase	+	10;	
					END_IF
					
					bHomingDone							:= FALSE;
				
				10: 
        	
					//Otwórz chwytaki
					bCapCatcher1				:= FALSE;
					bCapCatcher2				:= FALSE;
					bCapCatcher3				:= FALSE;
					bCapCatcher4				:= FALSE;
					//Wyłącz ssawki
					bCapSucker[1]					:= FALSE;
					bCapSucker[2]					:= FALSE;
					bCapSucker[3]					:= FALSE;
					bCapSucker[4]					:= FALSE;
					//Otwórz chwytaki słomek
					bStrawCatchersOpen			:= TRUE;
					bStrawCatchersClose			:= FALSE;
					//Cofnij chwytaki słomek
					bStrawCatcherActuatorIn		:= TRUE;
					bStrawCatcherActuatorOut	:= FALSE;
					//Podjedź robotem i chwytakiem słomek w górę jak cofnięty chwytak słomek - bazuj podnośnik Jisang
					IF tonStrawCatcherIn.Q THEN	
						mcCartesianZMoveAbsolute.Execute		:= TRUE;		
						mcCartesianZMoveAbsolute.Position		:= 420;//stParameters.lrTopZPosition;
						mcCartesianZMoveAbsolute.Acceleration	:= stParameters.lrPickerAcceleration;
						mcCartesianZMoveAbsolute.Deceleration	:= stParameters.lrPickerAcceleration;
						mcCartesianZMoveAbsolute.Velocity		:= 200;//stParameters.lrPickerSpeed;			
						
						fbStrawCatcherLift.bHoming;//				:= TRUE;
						//fbStrawCatcherLift.bHomingUp;//			:= TRUE;
						GVL_VIS.bCapSorterPreScrewerCatchStationHoming			:= NOT fbStrawCatcherLift.bHomingDone;
						GVL_VIS.bCapSorterPreScrewerCatcherStationHeightSet		:= NOT GVL_VIS.bCapSorterPreScrewerCatchStationHoming AND NOT bStrawCatcherLiftInHomePos;
						bEnableLift												:= TRUE;
						//Następny krok
						iHomingCase								:= iHomingCase + 10;
					END_IF
					//Reset komendy ruchu osi X
					mcCartesianYMoveAbsolute.Execute		:= FALSE;
					
			
				20:		
					(*Czekam na pozycję Z w górze i ruszam osią poziomą X na pozycję pobierania i czekam na obie pozycje*)
					bHomingWithoutJiesang						:= FALSE;
	    	
					IF (CartesianZAxisRef.NcToPlc.ActPos > stParameters.lrTopZPosition - stParameters.lrBendingDistance) OR
						mcCartesianZMoveAbsolute.Done THEN
						
						mcCatcherMoveAbsolute.Execute			:= TRUE;		
						mcCatcherMoveAbsolute.Position			:= stParameters.lrCatcherCatchingPosition;
						mcCatcherMoveAbsolute.Acceleration		:= stParameters.lrCatcherAcceleration;
						mcCatcherMoveAbsolute.Deceleration		:= stParameters.lrCatcherAcceleration;
						mcCatcherMoveAbsolute.Velocity			:= 30;//stParameters.lrCatcherSpeed;
						
						//Jedź osią poziomą Y na pozycję pick
						mcCartesianYMoveAbsolute.Execute		:= TRUE;
						mcCartesianYMoveAbsolute.Position		:= stParameters.lrPickYPosition;
						mcCartesianYMoveAbsolute.Acceleration	:= stParameters.lrPickerAcceleration;
						mcCartesianYMoveAbsolute.Deceleration	:= stParameters.lrPickerAcceleration;
						mcCartesianYMoveAbsolute.Velocity		:= 150;//stParameters.lrPickerSpeed;
						
						//Ustaw obracarkę w pozycji
						mcPreScrewerMoveRelative.Execute		:= TRUE;
						mcPreScrewerMoveRelative.Distance		:=  -1 * DINT_TO_LREAL(LREAL_TO_DINT(PreScrewerAxisRef.NcToPlc.SetPos) MOD 360);
						mcPreScrewerMoveRelative.Acceleration	:= stParameters.lrScrewAcceleration;
						mcPreScrewerMoveRelative.Deceleration	:= stParameters.lrScrewAcceleration;
						mcPreScrewerMoveRelative.Velocity		:= 180;//stParameters.lrScrewSpeed;
					END_IF
					IF mcPreScrewerMoveRelative.Done THEN
						mcPreScrewerMoveRelative.Execute		:= FALSE;
						mcPreScrewerHome(Axis := PreScrewerAxisRef, HomingMode := MC_Direct, Position := 0, Execute := TRUE);					
					END_IF
					//Jak obie pozycje osiągnięte to następny krok
					IF mcCartesianYMoveAbsolute.Done AND mcCartesianZMoveAbsolute.Done AND mcPreScrewerHome.Done AND bStrawCatcherLiftInHomePos THEN
						//Reset komendy ruchu osi
						bCapsBlowON								:= TRUE;
						bCapBlow1 								:= TRUE;
						bCapBlow2 								:= TRUE;
						bCapBlow3 								:= TRUE;
						bCapBlow4 								:= TRUE;
						mcCartesianYMoveAbsolute.Execute		:= FALSE;
						mcCartesianZMoveAbsolute.Execute		:= FALSE;
						mcPreScrewerHome.Execute				:= FALSE;
						//Reset homingu podnośnika Jisang
						fbStrawCatcherLift.bHoming;//				:= FALSE;
						GVL_VIS.bCapSorterPreScrewerCatchStationHoming			:= FALSE;
						GVL_VIS.bCapSorterPreScrewerCatcherStationHeightSet		:= FALSE;
					//	bEnableLift												:= FALSE;						
						
						
						//fbStrawCatcherLift.bHomingUp;//			:= FALSE;
						//Wysuń chwytaki słomek jesli to potrzebuje recepta
						bStrawCatcherActuatorIn					:= NOT stParameters.bStrawCatcherON;
						bStrawCatcherActuatorOut				:= stParameters.bStrawCatcherON;
						//Następny krok
						iHomingCase								:= iHomingCase + 10;
					END_IF
				
				30:	//Koniec
				IF NOT bCapBlow1 AND NOT bCapBlow2 AND NOT bCapBlow3 AND NOT bCapBlow4 THEN
						eState								:= E_Station.eHomingDone;
						bHomingDone							:= TRUE;
						iHomingCase							:= 0; 
				END_IF
				
				
				
				
				
				100://Odrzut nasadek
						//Otwórz chwytaki gdy nakrętka była zakręcana
					bCapCatcher1				R= bCapScrewed;
					bCapCatcher2				R= bCapScrewed;
					bCapCatcher3				R= bCapScrewed;
					bCapCatcher4				R= bCapScrewed;

						//Otwórz chwytaki słomek
					bStrawCatchersOpen			:= TRUE;
					bStrawCatchersClose			:= FALSE;
						//Cofnij chwytaki słomek
					bStrawCatcherActuatorIn		:= TRUE;
					bStrawCatcherActuatorOut	:= FALSE;
										//Podjedź robotem i chwytakiem słomek w górę jak cofnięty chwytak słomek - bazuj podnośnik Jisang
					IF tonStrawCatcherIn.Q THEN	
						mcCartesianZMoveAbsolute.Execute		:= TRUE;		
						mcCartesianZMoveAbsolute.Position		:= 420;//stParameters.lrTopZPosition;
						mcCartesianZMoveAbsolute.Acceleration	:= stParameters.lrPickerAcceleration;
						mcCartesianZMoveAbsolute.Deceleration	:= stParameters.lrPickerAcceleration;
						mcCartesianZMoveAbsolute.Velocity		:= 200;//stParameters.lrPickerSpeed;	70		
	
						//Następny krok
						iHomingCase								:= iHomingCase + 10;
					END_IF
					//Reset komendy ruchu osi X
					mcCartesianYMoveAbsolute.Execute		:= FALSE;
					
				110:
									(*Czekam na pozycję Z w górze i ruszam osią poziomą X na pozycję pobierania i czekam na obie pozycje*)
	    	
					IF (CartesianZAxisRef.NcToPlc.ActPos > stParameters.lrTopZPosition - stParameters.lrBendingDistance) OR
						mcCartesianZMoveAbsolute.Done THEN
						
						mcCatcherMoveAbsolute.Execute			:= TRUE;		
						mcCatcherMoveAbsolute.Position			:= stParameters.lrCatcherCatchingPosition;
						mcCatcherMoveAbsolute.Acceleration		:= stParameters.lrCatcherAcceleration;
						mcCatcherMoveAbsolute.Deceleration		:= stParameters.lrCatcherAcceleration;
						mcCatcherMoveAbsolute.Velocity			:= 200;//stParameters.lrCatcherSpeed;	70
						
						//Jedź osią poziomą Y na pozycję pick
						mcCartesianYMoveAbsolute.Execute		:= TRUE;
						mcCartesianYMoveAbsolute.Position		:= 3.0;
						mcCartesianYMoveAbsolute.Acceleration	:= stParameters.lrPickerAcceleration;
						mcCartesianYMoveAbsolute.Deceleration	:= stParameters.lrPickerAcceleration;
						mcCartesianYMoveAbsolute.Velocity		:= 200;//stParameters.lrPickerSpeed;	20
						
					END_IF
					
					//Jak obie pozycje osiągnięte to następny krok
					IF mcCartesianYMoveAbsolute.Done AND mcCartesianZMoveAbsolute.Done AND mcPreScrewerHome.Done AND fbStrawCatcherLift.bHomingDone THEN
						//Reset komendy ruchu osi

						mcCartesianYMoveAbsolute.Execute						:= FALSE;
						mcCartesianZMoveAbsolute.Execute						:= FALSE;
						mcPreScrewerHome.Execute								:= FALSE;
						//Reset homingu podnośnika Jisang
						fbStrawCatcherLift.bHoming;//				:= FALSE;
						GVL_VIS.bCapSorterPreScrewerCatchStationHoming			:= FALSE;
						GVL_VIS.bCapSorterPreScrewerCatcherStationHeightSet		:= FALSE;
						bEnableLift												:= FALSE;						
						//fbStrawCatcherLift.bHomingUp;//			:= FALSE;
						//Następny krok
						iHomingCase								:= iHomingCase + 10;
					END_IF		
					
					120:
					mcCartesianZMoveAbsolute.Execute			:= TRUE;		
					mcCartesianZMoveAbsolute.Position			:= 400;//stParameters.lrTopZPosition;
					mcCartesianZMoveAbsolute.Acceleration		:= stParameters.lrPickerAcceleration;
					mcCartesianZMoveAbsolute.Deceleration		:= stParameters.lrPickerAcceleration;
					mcCartesianZMoveAbsolute.Velocity			:= 200;//stParameters.lrPickerSpeed;	70
						
						IF mcCartesianZMoveAbsolute.Done THEN
							mcCartesianZMoveAbsolute.Execute	:= FALSE;	
								//Otwórz chwytaki
							bCapCatcher1						:= FALSE;
							bCapCatcher2						:= FALSE;
							bCapCatcher3						:= FALSE;
							bCapCatcher4						:= FALSE;
								//Wyłącz ssawki         		
							bCapSucker[1]							:= FALSE;
							bCapSucker[2]							:= FALSE;
							bCapSucker[3]							:= FALSE;
							bCapSucker[4]							:= FALSE;
							bCapsBlowON							:= TRUE;
							bCapBlow1 							:= TRUE;
							bCapBlow2 							:= TRUE;
							bCapBlow3 							:= TRUE;
							bCapBlow4 							:= TRUE;
							iHomingCase							:= iHomingCase + 10;
						END_IF
						
					130:
					IF NOT bCapBlow1 AND NOT bCapBlow2 AND NOT bCapBlow3 AND NOT bCapBlow4 THEN
						iHomingCase							:= 10; 
					END_IF
				
				
				
			END_CASE
		ELSE
			CASE iHomingCase OF
				0:
				mcCartesianYPower.Override					:=	100;			
				mcCartesianZPower.Override					:=	100;			
				mcPreScrewerPower.Override					:=	100;			
				mcCatcherPower.Override						:=	100;
				                                    		
				bCartesianYServoPower						:= TRUE;
				bCartesianZServoPower						:= TRUE;
				bPreScrewerPower							:= TRUE;
				bCatcherPower								:= TRUE;	
				                                    		
				mcCartesianYManualMove.JogBackwards			:=FALSE;
				mcCartesianZManualMove.JogBackwards			:=FALSE;
				mcPreScrewerManualMove.JogBackwards			:=FALSE;
				mcCatcherManualMove.JogBackwards			:=FALSE;
				                                    		
				mcCartesianYManualMove.JogForward			:=FALSE;
				mcCartesianZManualMove.JogForward			:=FALSE;
				mcPreScrewerManualMove.JogForward			:=FALSE;
				mcCatcherManualMove.JogForward				:=FALSE;
				bCycleNotDone								:= FALSE;
				iHomingCase									:= 10;
				bHomingDone									:= FALSE;
				
				10:
					//Otwórz chwytaki
				bCapCatcher1										:= FALSE;
				bCapCatcher2										:= FALSE;
				bCapCatcher3										:= FALSE;
				bCapCatcher4										:= FALSE;
				//Wyłącz ssawki             						
				bCapSucker[1]											:= FALSE;
				bCapSucker[2]											:= FALSE;
				bCapSucker[3]											:= FALSE;
				bCapSucker[4]											:= FALSE;
				//Otwórz chwytaki słomek    						
				bStrawCatchersOpen									:= TRUE;
				bStrawCatchersClose									:= FALSE;
				//Cofnij chwytaki słomek    						
				bStrawCatcherActuatorIn								:= TRUE;
				bStrawCatcherActuatorOut							:= FALSE;
				
					//Podjedź robotem i chwytakiem słomek w górę jak cofnięty chwytak słomek - bazuj podnośnik Jisang
					IF tonStrawCatcherIn.Q THEN	
						mcCartesianZMoveAbsolute.Execute				:= TRUE;		
						mcCartesianZMoveAbsolute.Position				:= 420;
						mcCartesianZMoveAbsolute.Acceleration			:= stParameters.lrPickerAcceleration;
						mcCartesianZMoveAbsolute.Deceleration			:= stParameters.lrPickerAcceleration;
						mcCartesianZMoveAbsolute.Velocity				:= 30;					                                     
						                                        		
						fbStrawCatcherLift.bHoming;//					:= TRUE;
						//fbStrawCatcherLift.bHomingUp;//					:= TRUE;
						GVL_VIS.bCapSorterPreScrewerCatchStationHoming			:= NOT fbStrawCatcherLift.bHomingDone;
						GVL_VIS.bCapSorterPreScrewerCatcherStationHeightSet		:= NOT GVL_VIS.bCapSorterPreScrewerCatchStationHoming AND NOT bStrawCatcherLiftInHomePos;
						bEnableLift												:= TRUE;
						//Następny krok
						iHomingCase										:= iHomingCase + 10;
					END_IF
				//Reset komendy ruchu osi X
				mcCartesianYMoveAbsolute.Execute					:= FALSE;
				
				20:
	(*Czekam na pozycję Z w górze i ruszam osią poziomą X na pozycję pobierania i czekam na obie pozycje*)
				bHomingWithoutJiesang						:= FALSE;
	
					IF (CartesianZAxisRef.NcToPlc.ActPos > stParameters.lrTopZPosition - stParameters.lrBendingDistance) OR
						mcCartesianZMoveAbsolute.Done THEN
						
						mcCatcherMoveAbsolute.Execute				:= TRUE;		
						mcCatcherMoveAbsolute.Position				:= stParameters.lrCatcherCatchingPosition;
						mcCatcherMoveAbsolute.Acceleration			:= stParameters.lrCatcherAcceleration;
						mcCatcherMoveAbsolute.Deceleration			:= stParameters.lrCatcherAcceleration;
						mcCatcherMoveAbsolute.Velocity				:= 30;
						                                            
							//Ustaw obracarkę w pozycji             
						mcPreScrewerMoveRelative.Execute			:= TRUE;
						mcPreScrewerMoveRelative.Distance			:=  -1 * DINT_TO_LREAL(LREAL_TO_DINT(PreScrewerAxisRef.NcToPlc.SetPos) MOD 360);
						mcPreScrewerMoveRelative.Acceleration		:= stParameters.lrScrewAcceleration;
						mcPreScrewerMoveRelative.Deceleration		:= stParameters.lrScrewAcceleration;
						mcPreScrewerMoveRelative.Velocity			:= 180;//stParameters.lrScrewSpeed;	
					END_IF			

					IF mcPreScrewerMoveRelative.Done AND mcCartesianZMoveAbsolute.Done AND 	fbStrawCatcherLift.bHomingDone THEN
						tonAxisYLagDetction.IN						:= FALSE;
						mcPreScrewerMoveRelative.Execute			:= FALSE;
						mcCatcherMoveAbsolute.Execute				:= FALSE;
						mcCartesianZMoveAbsolute.Execute			:= FALSE;
						iHomingCase									:= iHomingCase + 10;
					END_IF
				
				30:
				//Ustawiamy moment osi Y na 15%
				stAxisY_ADS.stCtr.uiNegativeTorqueLimit				:= 500;
				stAxisY_ADS.stCtr.uiPositiveTorqueLimit				:= 500; 
				uiAxisYTorqueLimit									:= 500;	
				mcCartesianYManualMove.JogForward					:= FALSE;
				mcCartesianYManualMove.JogBackwards					:= TRUE;
				mcCartesianYManualMove.Velocity						:= 5; 
				iHomingCase											:= iHomingCase + 10;
				
				40://Detekcja lag'a 
				tonAxisYLagDetction.IN								:= (ABS(CartesianYAxisRef.NcToPlc.PosDiff) >= 5.0);

					IF tonAxisYLagDetction.Q THEN
						mcCartesianYManualMove.JogBackwards			:= FALSE;
						iHomingCase									:= iHomingCase + 10;
					END_IF	
				
				50:
				mcCartesianYMoveRelative.Distance					:= 20;
				mcCartesianYMoveRelative.Execute					:= TRUE;
				
					IF mcCartesianYMoveRelative.Done THEN
						mcCartesianYMoveRelative.Execute			:= FALSE;
						iHomingCase									:= iHomingCase + 10;
					END_IF
				
				60:
				bCartesianYServoPower								:= FALSE;
				fbAxisYPositioningOffset.Position					:= 0;
				
					IF CartesianYAxisRef.Status.Disabled THEN
						iHomingCase									:= iHomingCase + 10;
					END_IF
					
				70:
				fbAxisYPositioningOffset.Execute					:= TRUE;
				
					IF 	fbAxisYPositioningOffset.Busy THEN
						iHomingCase									:= iHomingCase + 10;
					END_IF
				
				80:
				IF NOT fbAxisYPositioningOffset.Busy THEN	
					fbAxisYPositioningOffset.Execute				:= FALSE;
					bCartesianYServoPower							:= TRUE;
					stAxisY_ADS.stCtr.uiNegativeTorqueLimit			:= 2000;	//200%
					stAxisY_ADS.stCtr.uiPositiveTorqueLimit			:= 2000;	//200%
					iHomingCase										:= iHomingCase + 10;
				END_IF
				
				90:	
				bCapsBlowON											:= TRUE;
				bCapBlow1 											:= TRUE;
				bCapBlow2 											:= TRUE;
				bCapBlow3 											:= TRUE;
                bCapBlow4 											:= TRUE;
				iHomingCase											:= iHomingCase + 10;
				
				100://Oddmuch
				IF NOT bCapBlow1 AND NOT bCapBlow2 AND NOT bCapBlow3 AND NOT bCapBlow4 THEN
					iHomingCase										:= iHomingCase + 10;
				END_IF	
				
				110://Jedź osią poziomą Y na pozycję pick					
				mcCartesianYMoveAbsolute.Execute					:= TRUE;
				mcCartesianYMoveAbsolute.Position					:= stParameters.lrPickYPosition;
				mcCartesianYMoveAbsolute.Acceleration				:= stParameters.lrPickerAcceleration;
				mcCartesianYMoveAbsolute.Deceleration				:= stParameters.lrPickerAcceleration;
				mcCartesianYMoveAbsolute.Velocity					:= 30;//stParameters.lrPickerSpeed;
				
					IF mcCartesianYMoveAbsolute.Done THEN	//Koniec
						mcCartesianYMoveAbsolute.Execute			:= FALSE;
						eState										:= E_Station.eHomingDone;
						bHomingDone									:= TRUE;
						iHomingCase									:= 0; 
					END_IF	
					
			END_CASE
		END_IF
	END_IF
END_IF
END_ACTION

ACTION ManualMovements:
tonVacuumWatchdog(PT	:= stParameters.tTimeVacuumWatchdog);
trStepButton(CLK 		:= bStepButton OR (stCommandsIn.bPendantRightwardMovement AND diManualModeCase<>0));
rtSetEncoderOffsetAxisZ(CLK := bSetEncoderOffsetAxisZ);

// Wyjście z trybu manualnego
	IF NOT bManualMovement THEN		
		ResetCommands();		
		eState											:= E_Station.eReady;
	END_IF
	
	IF mcCartesianYManualMove.Done OR mcCartesianZManualMove.Done OR mcPreScrewerManualMove.Done OR mcCatcherManualMove.Done THEN
		bHomingDone										:= FALSE;
	END_IF

	//Zmiana prędkości plotera na kasecie sterowniczej
		rtPendantRightLeftFast(CLK 	:= stCommandsIn.bPendantRightLeftFast);
		ftPendantRightLeftFast(CLK 	:= stCommandsIn.bPendantRightLeftFast);	
		bChangeSpeedRightLeft 		S= (rtPendantRightLeftFast.Q OR ftPendantRightLeftFast.Q);	
		bChangeSpeedRightLeft 		R= NOT CartesianYAxisRef.Status.Moving;
		
		rtPendantUpDownFast(CLK 	:= stCommandsIn.bPendantUpDownFast);
		ftPendantUpDownFast(CLK 	:= stCommandsIn.bPendantUpDownFast);	
		bChangeSpeedUpDown			S= (rtPendantUpDownFast.Q OR ftPendantUpDownFast.Q);
		bChangeSpeedUpDown			R= NOT CartesianZAxisRef.Status.Moving;
	
 CASE 	diManualModeCase OF
	 
		 0:
	mcCatcherHalt.Execute								:=	FALSE;	 
		 
	 	//Ruchy manualne
	mcCartesianYManualMove.JogForward					:= NOT mcCartesianYManualMove.JogBackwards AND NOT bChangeSpeedRightLeft AND
															(bManualCartesianYJogPlus OR stCommandsIn.bPendantRightwardMovement);
	mcCartesianYManualMove.JogBackwards					:= NOT mcCartesianYManualMove.JogForward AND NOT bChangeSpeedRightLeft AND
															(bManualCartesianYJogMinus OR stCommandsIn.bPendantLeftwardMovement);
	mcCartesianYManualMove.Velocity						:= SEL(stCommandsIn.bPendantRightLeftFast, 5.0, 50.0); 
                                            			
	mcCartesianZManualMove.JogForward					:= NOT mcCartesianZManualMove.JogBackwards AND NOT bChangeSpeedUpDown AND
															(bManualCartesianZJogPlus OR stCommandsIn.bPendantUpwardMovement);
	mcCartesianZManualMove.JogBackwards					:= NOT mcCartesianZManualMove.JogForward AND NOT bChangeSpeedUpDown AND
															(bManualCartesianZJogMinus OR stCommandsIn.bPendantDownwardMovement);
	mcCartesianZManualMove.Velocity						:= SEL(stCommandsIn.bPendantUpDownFast, 5.0, 50.0); 
	                                        			
	mcPreScrewerManualMove.JogForward					:= bManualPreScrewerJogPlus;
	mcPreScrewerManualMove.JogBackwards					:= bManualPreScrewerJogMinus;
	mcPreScrewerManualMove.Velocity						:= 90;
                                            			
	mcCatcherManualMove.JogForward						:= bManualCatcherJogPlus;
	mcCatcherManualMove.JogBackwards					:= bManualCatcherJogMinus;
	mcCatcherManualMove.Velocity						:= 15; 
	                                        			
	bCapSucker[1]											:= bManualCapSucker1;	
	bCapSucker[2]											:= bmanualCapSucker2;	
	bCapSucker[3]											:= bManualCapSucker3;	
	bCapSucker[4]											:= bManualCapSucker4;	
	                          	    					                     
	bCapBlower1											:= bManualCapBlower1;	
	bCapBlower2											:= bManualCapBlower2;	
	bCapBlower3											:= bManualCapBlower3;	
	bCapBlower4											:= bManualCapBlower4;	
	                          		    				                 
	bCapCatcher1										:= bManualCapCatcher1;
	bCapCatcher2										:= bManualCapCatcher2;
	bCapCatcher3										:= bManualCapCatcher3;
	bCapCatcher4					    				:= bManualCapCatcher4;
	
	
	
	IF bManualStrawCatchersOpen	THEN
		bStrawCatchersOpen								:= TRUE;
		bStrawCatchersClose								:= FALSE;
		bManualStrawCatchersClose						:= FALSE;
	END_IF	                                    		
                                                		
	IF bManualStrawCatchersClose	THEN        		
		bStrawCatchersOpen								:= FALSE;
		bStrawCatchersClose								:= TRUE;
		bManualStrawCatchersOpen						:= FALSE;
	END_IF		                                		
	                                            		
     IF bManualStrawCatcherActuatorOut THEN     		
		 bStrawCatcherActuatorOut						:= TRUE;
		 bStrawCatcherActuatorIn						:= FALSE;
		 bManualStrawCatcherActuatorIn					:= FALSE;
	 END_IF                                     		
	                                            	
     IF bManualStrawCatcherActuatorIn THEN      	
		 bStrawCatcherActuatorIn						:= TRUE;
		 bStrawCatcherActuatorOut						:= FALSE;
		 bManualStrawCatcherActuatorOut					:= FALSE;
	 END_IF
	 
	 //Zaczynam sekwencje 
	 IF trStepButton.Q THEN
		 VirtualEna											:= TRUE;
		 ResetCommands();
		 bCapCatcher1										:= FALSE;
		 bCapCatcher2										:= false;
		 bCapCatcher3										:= false;
		 bCapCatcher4										:= false;
		 bCartesianReady									:= bCartesianInHomePos;
		 diManualModeCase									:= diManualModeCase + 10;
	 END_IF
	 
	 IF rtSetEncoderOffsetAxisZ.Q THEN
		diManualModeCase									:= diManualModeCase + 500;
	 END_IF
 
 
 		10:	//Dojazd do poz home
	bStepButton												:= TRUE;
	                                                    	
	mcCartesianZMoveAbsolute.Execute						:= NOT bAxisZInHomePos;		
	mcCartesianZMoveAbsolute.Position						:= 420;
	mcCartesianZMoveAbsolute.Acceleration					:= 200.0;
	mcCartesianZMoveAbsolute.Deceleration					:= 200.0;
	mcCartesianZMoveAbsolute.Velocity						:= 30;
	                                        				
	//najpierw os Z potem winda chwytakow   				
	mcCatcherMoveAbsolute.Execute							:= NOT bAxisStrawCatcherHomePos AND bAxisZInHomePos;		
	mcCatcherMoveAbsolute.Position							:= stParameters.lrCatcherCatchingPosition;
	mcCatcherMoveAbsolute.Acceleration						:= 200.0;
	mcCatcherMoveAbsolute.Deceleration						:= 200.0;
	mcCatcherMoveAbsolute.Velocity							:= 30;
	                                        				
	mcCartesianYMoveAbsolute.Execute						:= NOT bAxisYInHomePos AND bAxisZInHomePos;
	mcCartesianYMoveAbsolute.Position						:= stParameters.lrPickYPosition;
	mcCartesianYMoveAbsolute.Acceleration					:= 200.0;
	mcCartesianYMoveAbsolute.Deceleration					:= 200.0;
	mcCartesianYMoveAbsolute.Velocity						:= 30; 
	                                                    	
	IF bAxisZInHomePos THEN
		GVL_VIS.bCapSorterPreScrewerCatchStationHoming			:= NOT fbStrawCatcherLift.bHomingDone;
		GVL_VIS.bCapSorterPreScrewerCatcherStationHeightSet		:= NOT GVL_VIS.bCapSorterPreScrewerCatchStationHoming AND NOT bStrawCatcherLiftInHomePos;
		bEnableLift												:= GVL_VIS.bCapSorterPreScrewerCatcherStationHeightSet;
	END_IF

		IF 	bCartesianInHomePos AND bStrawCatcherLiftInHomePos THEN
			mcCartesianZMoveAbsolute.Execute              	:= FALSE;
			mcCatcherMoveAbsolute.Execute                 	:= FALSE;
			mcCartesianYMoveAbsolute.Execute              	:= FALSE;
			GVL_VIS.bCapSorterPreScrewerCatchStationHoming	:= FALSE;
			diManualModeCase								:= diManualModeCase + 5;
		END_IF
		
		15: //Ustaw obracarkę w pozycji
	bStepButton												:= TRUE;
	                                                    	
	mcPreScrewerMoveRelative.Execute						:= TRUE;
	mcPreScrewerMoveRelative.Distance						:=  -1 * DINT_TO_LREAL(LREAL_TO_DINT(PreScrewerAxisRef.NcToPlc.SetPos) MOD 360);
	mcPreScrewerMoveRelative.Acceleration					:= 200.0;
	mcPreScrewerMoveRelative.Deceleration					:= 200.0;
	mcPreScrewerMoveRelative.Velocity						:= 180.0;	
	                                                    	
		IF mcPreScrewerMoveRelative.Done THEN           	
			mcPreScrewerMoveRelative.Execute				:= FALSE;
			
			IF bCartesianReady THEN
				diManualModeCase							:= diManualModeCase + 10;
			ELSE	                                        
				bStepButton									:= FALSE;
				diManualModeCase							:= diManualModeCase + 5;
			END_IF
			
		END_IF	

		
//--------------------------------jazda na poz pick------------------------------------------------------------------			
		20:	//Kolejny krok
	 IF trStepButton.Q THEN
		diManualModeCase									:= diManualModeCase + 5;
	 END_IF

		25:
	bStepButton												:= TRUE;
	
	mcCartesianZMoveAbsolute.Execute						:= TRUE;		
	mcCartesianZMoveAbsolute.Position						:= stParameters.lrPickZPosition;
	
		IF mcCartesianZMoveAbsolute.Done THEN
			mcCartesianZMoveAbsolute.Execute				:= FALSE;
			bStepButton										:= FALSE;
			diManualModeCase								:= diManualModeCase + 5;
		END_IF

		
//----------------------------Sekwencyjne zalączanie ssawek----------------------------------------------------------------	
		30: //Kolejny krok
	 IF trStepButton.Q THEN
		FOR i:=1 TO 4 DO
			bCapSucker[i]									:= TRUE;
		END_FOR	 
	 
		diManualModeCase									:= diManualModeCase + 5;
	 END_IF
		
		35: //Załączanie ssawek
	tonVacuumWatchdog.IN									:= TRUE;
	bStepButton												:= TRUE;

	
	
		IF tonVacuumWatchdog.Q THEN	
			bStepButton										:= FALSE;		 
			tonVacuumWatchdog.IN							:= FALSE;								
			diManualModeCase								:= diManualModeCase + 20;				
		END_IF
		
		
//-------------------------------Dojazd do pozycji zamykania wings'ów-------------------------------------------------------------------			
		55: //Kolejny krok
	 IF trStepButton.Q THEN
		diManualModeCase									:= diManualModeCase + 5;
	 END_IF	
	 
	 	60:
	bStepButton												:= TRUE;	
	mcCartesianZMoveAbsolute.Execute						:= TRUE;		
	mcCartesianZMoveAbsolute.Position						:= stParameters.lrCapCatcherZPosition;	
		
		IF mcCartesianZMoveAbsolute.Done THEN
			
			FOR i:=1 TO 4 DO
				bCapSucker[i]								R= NOT  bCapSucker[i];
			END_FOR 
			
			bStepButton										:= FALSE;	
			mcCartesianZMoveAbsolute.Execute				:= FALSE;
			diManualModeCase								:= diManualModeCase + 5;		
		END_IF

		
//--------------------------------Zamykanie vings'ów------------------------------------------------------------------			
		65://Kolejny krok
	 IF trStepButton.Q THEN
		diManualModeCase									:= diManualModeCase + 5;
	 END_IF	
	 
	 	70:
	bStepButton												:= FALSE;	
	bCapCatcher1											:= TRUE;
	bCapCatcher2											:= TRUE;
	bCapCatcher3											:= TRUE;
	bCapCatcher4											:= TRUE;
	diManualModeCase										:= diManualModeCase + 5;

	
//---------------------------------dojazd do poz. Top-----------------------------------------------------------------			
		75://Kolejny krok
	 IF trStepButton.Q THEN
		diManualModeCase									:= diManualModeCase + 5;
	 END_IF	
		
		80:
	bStepButton												:= TRUE;
	mcCartesianZMoveAbsolute.Execute						:= TRUE;
	mcCartesianZMoveAbsolute.Position						:= stParameters.lrTopZPosition;
		
		IF mcCartesianZMoveAbsolute.Done THEN
			bStepButton										:= FALSE;	
			mcCartesianZMoveAbsolute.Execute				:= FALSE;
			diManualModeCase								:= diManualModeCase + 5;		
		END_IF

		
//-----------------------------------dojazd osi Y do pozycji place---------------------------------------------------------------			
		85://Kolejny krok
	 IF trStepButton.Q THEN
		diManualModeCase									:= diManualModeCase + 5;
	 END_IF	
	 
	 90:
	bStepButton												:= TRUE;
	mcCartesianYMoveAbsolute.Execute						:= TRUE;
	mcCartesianYMoveAbsolute.Position						:= stParameters.lrPlaceYPosition;
	
	 mcCartesianZMoveAbsolute.Execute						:= CartesianYAxisRef.NcToPlc.ActPos > stParameters.lrPickYPosition + 50.0;
	 mcCartesianZMoveAbsolute.Position						:= stParameters.lrCartesianCatchZPosition;
	 
		IF mcCartesianYMoveAbsolute.Done AND mcCartesianZMoveAbsolute.Done THEN
			bStepButton										:= FALSE;
			mcCartesianYMoveAbsolute.Execute				:= FALSE;
			GVL_VIS.bCapSorterPreScrewerBottleCatcherCatch	:= TRUE;					//Zamykanie chwytaków butelek
			diManualModeCase								:= diManualModeCase + 10;
		END_IF		
		
		
		
		

		
//-------------------------------Wybór pracy: słomka albo fliptop & sterowanie krabami------------------------	
		100://Kolejny krok
	 IF trStepButton.Q THEN
		diManualModeCase									:= diManualModeCase + 5;
	 END_IF	
	 
		105://Ustaw pozycję wirtualnej osi tak samo jak na osi Z
	fbVirtualAxis.fPosition									:= CartesianZAxisRef.NcToPlc.ActPos;
	fbVirtualAxis.SetPosAbsClearLag(bExecute				:= TRUE);
		
		IF fbVirtualAxis.pSetPos.Busy THEN
			diManualModeCase								:= diManualModeCase + 1;
		ELSIF fbVirtualAxis.pSetPos.Error OR fbVirtualAxis.pSetPos.CommandAborted THEN
    		udiErrorID										:= 6;
    		udiErrorID										:= udiErrorID + iStationIndex;
    		sErrorDescription								:= 'Błąd podnosnika lub brak zasilania';
    		sErrorDescription2								:= ' ';	
		END_IF
		
		106:
	fbVirtualAxis.SetPosAbsClearLag(bExecute				:= FALSE);
		
		IF fbVirtualAxis.pSetPos.Done THEN
			diManualModeCase								:= diManualModeCase + 4;
		END_IF


		110: 	//Przy aktywowanych slomkach--> wysuń kraby
	IF stParameters.bStrawCatcherON THEN
		bStrawCatcherActuatorIn								:= FALSE;
		bStrawCatcherActuatorOut							:= TRUE; 
		diManualModeCase									:= diManualModeCase + 1;
	ELSE
			//przeskakuję do sprawdzania czy mam szukanie gwintu
		bStrawCatcherActuatorIn								:= TRUE;
		bStrawCatcherActuatorOut							:= FALSE; 			
		fbGearInAxisZ.Enable								:= TRUE;
		
			IF fbGearInAxisZ.InGear THEN
				fbGearInAxisZ.Enable						:= FALSE;
				IF stParameters.lrScrewFinding > 0 THEN
			 		diManualModeCase						:= diManualModeCase + 26;
		 		ELSE
					diManualModeCase						:= diManualModeCase + 30;
			 	END_IF
			 END_IF
	END_IF
		
		
		111://zamknij kraby
	bStepButton												:= TRUE;	
	bStrawCatchersOpen										:= NOT bStrawCatcherOut;
	bStrawCatchersClose										:= bStrawCatcherOut;
	
		//zamkniete kraby
		IF tonStrawCatcher1Close.Q (*AND tonStrawCatcher2Close.Q*) AND tonStrawCatcher3Close.Q AND tonStrawCatcher4Close.Q THEN
			bStepButton										:= FALSE;
			diManualModeCase								:= diManualModeCase + 4;
		END_IF

		
//-----------------------------------Prowadzenie slomki do pozycji wspolnego ruchu-------------------------------			
		115://Kolejny krok
	 IF trStepButton.Q THEN
		diManualModeCase									:= diManualModeCase + 5;
	 END_IF			
		
		120://gear'owanie napędu prowadzenia słomki
	fbGearInCatcherAxis.Enable								:= TRUE;
	fbGearInCatcherAxis.GearRatio							:= 1;
	fbGearInAxisZ.Enable									:= TRUE;
	fbGearInAxisZ.GearRatio									:= 0.0000000001;
	bStepButton												:= TRUE;
		
		IF fbGearInCatcherAxis.InGear AND fbGearInAxisZ.InGear THEN
			//fbGearInCatcherAxis.Enable						:= FALSE;
			//fbGearInAxisZ.Enable							:= FALSE;
			diManualModeCase								:= diManualModeCase + 10;
		END_IF

		
//-----------------------------------Prowadzenie, wkładanie nasadki oraz rozgirowanie osi do prowadzenia słomki------------------------------------------			
		130: 
	fbVirtualAxis.fPosition									:= (stParameters.LrCheckStrawCatcherActuatorZPosition - stParameters.lrStrawInsertDistance);	//Pozycja sprawdzania cofnięcia krabów
	fbVirtualAxis.fVelocity									:= 100.0;	//10
	fbVirtualAxis.fAcceleration								:= 1000.0;
	fbVirtualAxis.fDeceleration								:= 1000.0;
	fbVirtualAxis.fJerk										:= 10000.0;			
			
	bStepButton												:= TRUE;
	bVirtualMove											:= TRUE;				
//	fbGearInAxisZ.Execute									:= CatcherAxisRef.NcToPlc.ActPos <= (stParameters.lrCatcherPlacePosition + stParameters.lrStrawInsertDistance);

	//IF CatcherAxisRef.NcToPlc.ActPos <= (stParameters.lrCatcherCatchingPosition - stParameters.lrStrawInsertDistance) THEN
	//	fbGearInAxisZ.GearRatio								:= 1;
	//END_IF
	
	IF (CatcherAxisRef.NcToPlc.ActPos + stParameters.lrCatcherHightSV) <= (stParameters.lrCartesianCatchZPosition-(stParameters.lrCapHight + 25)) THEN
		fbGearInAxisZ.GearRatio								:= 1;
	END_IF
	
			//Otwórz chwytaki słomek
		IF CartesianZAxisRef.NcToPlc.ActPos <= stParameters.lrStrawCatcherZPosition THEN					
			bStrawCatchersOpen								:= TRUE;
			bStrawCatchersClose								:= FALSE;
		END_IF
		
		// 10mm stały offset - wysokość nad butelką
		IF (CatcherAxisRef.NcToPlc.ActPos <= 1.0) OR (CatcherAxisRef.NcToPlc.ActPos + 32 <= ((stParameters.lrBottleHight + 10.0) - stParameters.lrCatcherHightSV)) THEN	//13 20
			fbGearInCatcherAxis.GearRatio					:= 0.0000000001;
		END_IF
	
			IF tonStrawCatcher1Open.Q AND tonStrawCatcher2Open.Q AND tonStrawCatcher3Open.Q AND tonStrawCatcher4Open.Q THEN																				
				//Cofnij chwytaki słomek
				bStrawCatcherActuatorIn						:= TRUE;
				bStrawCatcherActuatorOut					:= FALSE;				
			END_IF			
			
				IF stVirtualMove_Out.Done THEN
					//fbGearInAxisZ.Enable					:= FALSE;
					//fbGearOutCatcherAxis.Execute			:= FALSE;
					fbGearInCatcherAxis.GearRatio				:= 0.0000000001;
					bVirtualMove							:= FALSE;	
					bStepButton								:= FALSE;
					diManualModeCase						:= diManualModeCase + 5;
				END_IF					
		
//------------------------------------Zakończenie wkładania nasadki---------------------------------------------------			
		135://Kolejny krok
		//mcCatcherHalt.Execute								:=	FALSE;
		
	 IF trStepButton.Q THEN
		 IF stParameters.lrScrewFinding > 0 THEN
			 diManualModeCase								:= diManualModeCase + 1;
		 ELSE
			 diManualModeCase								:= diManualModeCase + 5;
		 END_IF
		
	 END_IF	

//------------------------------------Szukanie gwintu---------------------------------------------------				 	
		136:
	fbVirtualAxis.fVelocity									:= 800.0;	//10
	fbVirtualAxis.fAcceleration								:= 1000.0;
	fbVirtualAxis.fDeceleration								:= 1000.0;
	fbVirtualAxis.fJerk										:= 10000.0;			
		
	fbVirtualAxis.fPosition									:= stParameters.lrScrewerStartZPosition;
	bVirtualMove											:= TRUE;
	bStepButton												:= TRUE;	
	
		IF stVirtualMove_Out.Done THEN
			bCapSucker[1]										:= FALSE;
			bCapSucker[2]										:= FALSE;
			bCapSucker[3]										:= FALSE;
			bCapSucker[4]										:= FALSE;

			mcPreScrewerMoveRelative.Distance				:= stParameters.lrScrewFinding * -1.0;
			mcPreScrewerMoveRelative.Acceleration			:= stParameters.lrScrewAcceleration;
			mcPreScrewerMoveRelative.Deceleration			:= stParameters.lrScrewAcceleration;
			mcPreScrewerMoveRelative.Velocity				:= stParameters.lrScrewSpeed;
			mcPreScrewerMoveRelative.Execute				:= TRUE;
		END_IF
		
				IF mcPreScrewerMoveRelative.Done OR ABS(PreScrewerAxisRef.NcToPlc.PosDiff) > 60.0 OR mcPreScrewerMoveRelative.Error THEN
					bVirtualMove							:= FALSE;
					bStepButton								:= FALSE;
					mcPreScrewerMoveRelative.Execute		:= FALSE;
					diManualModeCase						:= diManualModeCase + 1;
				END_IF	
		
		137://Kolejny krok
	 IF trStepButton.Q THEN
		 diManualModeCase									:= diManualModeCase + 3;		
	 END_IF					
	 
	 	140:
	lrPreScrewerAxisSavedPosition							:= PreScrewerAxisRef.NcToPlc.ActPos;	//zapisywanie pozycji przed zakrecaniem		
	fbVirtualAxis.fPosition									:= stParameters.lrPlaceZPosition - stParameters.lrStrawInsertDistance;
	fbVirtualAxis.fVelocity									:= stParameters.lrCatcherSpeed;
	fbVirtualAxis.fAcceleration								:= 1000.0;
	fbVirtualAxis.fDeceleration								:= 1000.0;
	fbVirtualAxis.fJerk										:= 10000.0;
	bVirtualMove											:= TRUE;
	bStepButton												:= TRUE;
	
		IF CartesianZAxisRef.NcToPlc.ActPos <= stParameters.lrScrewerStartZPosition + 1.0 THEN
			bCapSucker[1]										:= FALSE;
			bCapSucker[2]										:= FALSE;
			bCapSucker[3]										:= FALSE;
			bCapSucker[4]										:= FALSE;
			mcPreScrewerMoveRelative.Execute				:= TRUE;
			mcPreScrewerMoveRelative.Distance				:= stParameters.lrScrewDistance;
			mcPreScrewerMoveRelative.Acceleration			:= stParameters.lrScrewAcceleration;
			mcPreScrewerMoveRelative.Deceleration			:= stParameters.lrScrewAcceleration;
			mcPreScrewerMoveRelative.Velocity				:= stParameters.lrScrewSpeed;// do bylo 600.0;//stParameters.lrScrewSpeed;
			diManualModeCase								:= diManualModeCase + 5;			
		END_IF

	
		145:
	bStepButton												:= TRUE;
	
			//otwórz centrowniki butelek
		IF (GVL_Recipe.bCapSorterPreScrewerCatchAngleOpenEnaShow AND
			ABS(PreScrewerAxisRef.NcToPlc.ActPos - lrPreScrewerAxisSavedPosition) >= GVL_Recipe.lrCapSorterPreScrewerCatchAngleOpenSV) THEN
			bBottleCatcherCatchTemp					:= FALSE;
		END_IF
	
		IF PreScrewerAxisRef.NcToPlc.PosDiff > 100.0 OR (stVirtualMove_Out.Done AND mcPreScrewerMoveRelative.Done) THEN
			bBottleCatcherCatchTemp							:= FALSE;
			bCapCatcher1									:= FALSE;
		 	bCapCatcher2									:= FALSE;
		 	bCapCatcher3									:= FALSE;
		 	bCapCatcher4									:= FALSE;
			bVirtualMove									:= FALSE;
			bCapsBlowON										:= TRUE;
			
				IF fbVirtualAxis.bMoving THEN
					fbVirtualAxis.Halt(bExecute := TRUE);
				ELSE
					fbVirtualAxis.Halt(bExecute := FALSE);
					diManualModeCase						:= diManualModeCase + 5;
				END_IF	
				
		END_IF
		
		150:
	bStepButton												:= TRUE;	
	fbVirtualAxis.fPosition									:= stParameters.lrPlaceZPosition + 20.0;	
	fbVirtualAxis.fVelocity									:= 800.0;//10.0;
	fbVirtualAxis.fAcceleration								:= 1000.0;
	fbVirtualAxis.fDeceleration								:= 1000.0;
	fbVirtualAxis.fJerk										:= 10000.0;
	bVirtualMove											:= TRUE;
	fbGearInCatcherAxis.Enable								:= FALSE;
	fbGearInAxisZ.Enable									:= FALSE;
	
		IF stVirtualMove_Out.Done THEN
			bVirtualMove									:= FALSE;
			diManualModeCase								:= diManualModeCase + 5;
		END_IF
		
		
					151:		//na testy do usunięcia
					fbVirtualAxis.fPosition									:= CartesianZAxisRef.NcToPlc.ActPos;
					fbVirtualAxis.SetPosAbsClearLag(bExecute				:= TRUE);
					
					152:
					fbVirtualAxis.SetPosAbsClearLag(bExecute				:= FALSE);
	
	
		155:
	fbGearOutAxisZ.Execute									:= TRUE;
	fbGearOutCatcherAxis.Execute							:= TRUE;
	
		IF NOT CartesianZAxisRef.Status.Coupled AND NOT CatcherAxisRef.Status.Coupled THEN
			fbGearOutAxisZ.Execute							:= FALSE;
			fbGearOutCatcherAxis.Execute					:= FALSE;
			bStepButton										:= FALSE;
			diManualModeCase								:= diManualModeCase + 5;
		END_IF

//-------------------------------------Dojazd do poz home---------------------------------------------			
		160://Kolejny krok
	 IF trStepButton.Q THEN
		diManualModeCase									:= diManualModeCase + 5;
	 END_IF	
		
		165:
	GVL_VIS.bCapSorterPreScrewerBottleCatcherCatch	:= FALSE;	
	bStepButton										:= TRUE;	
	mcCartesianZMoveAbsolute.Execute				:= TRUE;		
	mcCartesianZMoveAbsolute.Position				:= stParameters.lrTopZPosition;
                                            		
	mcCartesianYMoveAbsolute.Execute				:= ABS(mcCartesianZMoveAbsolute.Position - stParameters.lrTopZPosition) <= 1.0;
	mcCartesianYMoveAbsolute.Position				:= stParameters.lrPickYPosition;
	                                        		
	mcPreScrewerMoveRelative.Execute				:= mcCartesianYMoveAbsolute.Done;
	mcPreScrewerMoveRelative.Velocity				:= 180.0;
	mcPreScrewerMoveRelative.Distance				:= -1 * DINT_TO_LREAL(LREAL_TO_DINT(PreScrewerAxisRef.NcToPlc.SetPos) MOD 360);
	                                        		
	mcCatcherMoveAbsolute.Execute					:= mcCartesianZMoveAbsolute.Done;		
	mcCatcherMoveAbsolute.Position					:= stParameters.lrCatcherCatchingPosition;
	
		IF (mcCartesianZMoveAbsolute.Done AND mcCartesianYMoveAbsolute.Done
			AND mcPreScrewerMoveRelative.Done AND mcCatcherMoveAbsolute.Done) THEN
				bCapsBlowON							:= TRUE;
				bStepButton							:= FALSE;
				ResetCommands();            		
				diManualModeCase					:= 0;
		END_IF	 
		
		
	500: //Ustawianie offsetu na soi Z kartezjana
	bCartesianZServoPower				:= FALSE;
	
	fbAxisZPositioningOffset.Position	:= 0.0;
	fbAxisZPositioningOffset.Execute	:= NOT CartesianZAxisRef.Status.Disabled;
	
	IF fbAxisZPositioningOffset.Busy THEN
		diManualModeCase				:= diManualModeCase + 5;
	END_IF
		
	505:
	IF NOT fbAxisZPositioningOffset.Busy THEN
		fbAxisZPositioningOffset.Execute := FALSE;
		bCartesianZServoPower			 := TRUE;
		diManualModeCase				:= diManualModeCase + 5;
	END_IF
	
	510:
	IF 	mcCartesianZPower.Status THEN
		diManualModeCase				:= 0;
	END_IF
		
 END_CASE
END_ACTION

ACTION PreparingToDisable:
//BAZOWANIE 

mcCartesianYPower.Override				:=	100;			
mcCartesianZPower.Override				:=	100;			
mcPreScrewerPower.Override				:=	100;			
mcCatcherPower.Override					:=	100;	

bCartesianYServoPower					:= TRUE;
bCartesianZServoPower					:= TRUE;
bPreScrewerPower						:= TRUE;
bCatcherPower							:= TRUE;	

mcCartesianYManualMove.JogBackwards		:=FALSE;
mcCartesianZManualMove.JogBackwards		:=FALSE;
mcPreScrewerManualMove.JogBackwards		:=FALSE;
mcCatcherManualMove.JogBackwards		:=FALSE;

mcCartesianYManualMove.JogForward		:=FALSE;
mcCartesianZManualMove.JogForward		:=FALSE;
mcPreScrewerManualMove.JogForward		:=FALSE;
mcCatcherManualMove.JogForward			:=FALSE;
bCycleNotDone							:= FALSE;



IF mcCartesianYPower.Status AND mcCartesianZPower.Status AND mcPreScrewerPower.Status AND mcCatcherPower.Status THEN
		
		CASE iDisablingCase OF
		
			0:
				iDisablingCase							:= iDisablingCase	+	10;
			
			10: 

				//Otwórz chwytaki
				bCapCatcher1				:= FALSE;
				bCapCatcher2				:= FALSE;
				bCapCatcher3				:= FALSE;
				bCapCatcher4				:= FALSE;
				//Wyłącz ssawki
				bCapSucker[1]				:= FALSE;
				bCapSucker[2]				:= FALSE;
				bCapSucker[3]				:= FALSE;
				bCapSucker[4]				:= FALSE;
				//Wyłącz odmuchy
				bCapBlower1					:= FALSE;
				bCapBlower2					:= FALSE;
				bCapBlower3					:= FALSE;
				bCapBlower4					:= FALSE;
				//Otwórz chwytaki słomek
				bStrawCatchersOpen			:= TRUE;
				bStrawCatchersClose			:= FALSE;
				//Cofnij chwytaki słomek
				bStrawCatcherActuatorIn		:= TRUE;
				bStrawCatcherActuatorOut	:= FALSE;
				//Podjedź robotem i chwytakiem słomek w górę jak cofnięty chwytak słomek - bazuj podnośnik Jisang
				IF tonStrawCatcherIn.Q THEN	
					mcCartesianZMoveAbsolute.Execute		:= TRUE;		
					mcCartesianZMoveAbsolute.Position		:= 420;//stParameters.lrTopZPosition;
					mcCartesianZMoveAbsolute.Acceleration	:= stParameters.lrPickerAcceleration;
					mcCartesianZMoveAbsolute.Deceleration	:= stParameters.lrPickerAcceleration;
					mcCartesianZMoveAbsolute.Velocity		:= 30;//stParameters.lrPickerSpeed;
					
					mcCatcherMoveAbsolute.Execute			:= TRUE;		
					mcCatcherMoveAbsolute.Position			:= stParameters.lrCatcherCatchingPosition;
					mcCatcherMoveAbsolute.Acceleration		:= stParameters.lrCatcherAcceleration;
					mcCatcherMoveAbsolute.Deceleration		:= stParameters.lrCatcherAcceleration;
					mcCatcherMoveAbsolute.Velocity			:= 30;//stParameters.lrCatcherSpeed;

					//Następny krok
					iDisablingCase								:= iDisablingCase + 10;
				END_IF
				//Reset komendy ruchu osi X
				mcCartesianYMoveAbsolute.Execute		:= FALSE;
				
		
			20:		
	(*Czekam na pozycję Z w górze i ruszam osią poziomą X na pozycję pobierania i czekam na obie pozycje*)
				//bStrawCatcherLiftEnable						R= ABS(CartesianYAxisRef.NcToPlc.ActPos - stParameters.lrPickYPosition)<=10.0;
				
				IF (CartesianZAxisRef.NcToPlc.ActPos > stParameters.lrTopZPosition - stParameters.lrBendingDistance) OR
					mcCartesianZMoveAbsolute.Done THEN					
					//Jedź osią poziomą X na pozycję pick
					mcCartesianYMoveAbsolute.Execute		:= TRUE;
					mcCartesianYMoveAbsolute.Position		:= stParameters.lrPickYPosition;
					mcCartesianYMoveAbsolute.Acceleration	:= stParameters.lrPickerAcceleration;
					mcCartesianYMoveAbsolute.Deceleration	:= stParameters.lrPickerAcceleration;
					mcCartesianYMoveAbsolute.Velocity		:= 30;//stParameters.lrPickerSpeed;
					//Ustaw obracarkę w pozycji
					mcPreScrewerMoveRelative.Execute		:= TRUE;
					mcPreScrewerMoveRelative.Distance		:=  -1 * DINT_TO_LREAL(LREAL_TO_DINT(PreScrewerAxisRef.NcToPlc.SetPos) MOD 360);
					mcPreScrewerMoveRelative.Acceleration	:= stParameters.lrScrewAcceleration;
					mcPreScrewerMoveRelative.Deceleration	:= stParameters.lrScrewAcceleration;
					mcPreScrewerMoveRelative.Velocity		:= 180;//stParameters.lrScrewSpeed;
				END_IF
				IF mcPreScrewerMoveRelative.Done THEN
					mcPreScrewerMoveRelative.Execute		:= FALSE;
					mcPreScrewerHome(Axis := PreScrewerAxisRef, HomingMode := MC_Direct, Position := 0, Execute := TRUE);					
				END_IF
				//Jak obie pozycje osiągnięte to następny krok
				IF mcCartesianYMoveAbsolute.Done AND mcCartesianZMoveAbsolute.Done AND mcPreScrewerHome.Done AND fbStrawCatcherLift.eState =  E_Station.eDisabled THEN
					//Reset komendy ruchu osi
					mcCartesianYMoveAbsolute.Execute		:= FALSE;
					mcCartesianZMoveAbsolute.Execute		:= FALSE;
					mcPreScrewerHome.Execute				:= FALSE;
					//Wysuń chwytaki słomek jesli to potrzebuje recepta
					bStrawCatcherActuatorIn					:= TRUE;
					bStrawCatcherActuatorOut				:= FALSE;
					//Następny krok
					iDisablingCase								:= iDisablingCase + 10;
				END_IF
			
			30:	//Koniec
				eState								:= E_Station.eDisabled;
				bHomingDone							:= FALSE;
				iDisablingCase						:= 0;
		END_CASE
END_IF
END_ACTION

ACTION Reject:

CASE iRejectCase OF
	0:

		mcCartesianZMoveAbsolute.Position	:= stParameters.lrPickZPosition - lrAxisZ_RejectOffset;	
		mcCartesianZMoveAbsolute.Execute	:= NOT bTubeReject;
	
				//Przyssanie wszystkich nasadek (przypadek wcisnietej), lub pojedynczej (wykryto brak słomki)
			FOR i:=1 TO 4 DO	
				bCapSucker[i]					:=SEL(bTubeReject, stParameters.bPickerActiv[i] AND NOT tonSuckedOk[i].Q, NOT stMoverStatus.stSlotStatus[i].bTubePresent AND stParameters.bPickerActiv[i]);//SEL(bTubeReject, TRUE, NOT stMoverStatus.stSlotStatus[i].bTubePresent AND stParameters.bPickerActiv[i]);
			END_FOR
		
		iRejectCase	:= 5;
	
	
	5:
			IF bTubeReject OR mcCartesianZMoveAbsolute.Done THEN
				mcCartesianZMoveAbsolute.Execute	:= FALSE;
				iRejectCase	:= 10;
			END_IF
	
	10:
		tonVacuumWatchdog.IN					:= TRUE;
	

		
			IF bAllSlotsVacuumStatus OR tonVacuumWatchdog.Q THEN
					//Podjazd do góry
				mcCartesianZMoveAbsolute.Position	:= stParameters.lrTopZPosition;
				mcCartesianZMoveAbsolute.Execute	:= TRUE;	
				tonVacuumWatchdog.IN				:= FALSE;
				iRejectCase	:= 20;
			END_IF
	
	20:
			//Zamykanie łapek
			IF CartesianZAxisRef.NcToPlc.ActPos > stParameters.lrCapCatcherZPosition THEN
				bCapCatcher1					:= TRUE;
				bCapCatcher2					:= TRUE;
				bCapCatcher3					:= TRUE;
				bCapCatcher4					:= TRUE;
			ELSIF rtAxisZMoving.Q THEN	//oddmuch nie przyssanych nakrętek
				bCapBlow1						:= NOT bCapSucker[1];
            	bCapBlow2						:= NOT bCapSucker[2];
            	bCapBlow3						:= NOT bCapSucker[3];
            	bCapBlow4						:= NOT bCapSucker[4];
				bCapsBlowON						:= TRUE;
			END_IF
			
			IF ABS(CartesianZAxisRef.NcToPlc.ActPos - mcCartesianZMoveAbsolute.Position) <= stParameters.lrBendingDistance THEN
				mcCartesianZMoveAbsolute.Execute	:= FALSE;	
				bMissingCaps						:= TRUE;
				mcCartesianYMoveAbsolute.Position	:= 3.0;
				mcCartesianYMoveAbsolute.Execute	:= TRUE;
				
					FOR i:= 1 TO 4 DO
						bCapSucker[i]				:= FALSE;
					END_FOR				
				
				iRejectCase							:= 30;
			END_IF
		
		30:
			IF ABS(CartesianYAxisRef.NcToPlc.ActPos - mcCartesianYMoveAbsolute.Position) <= stParameters.lrBendingDistance THEN
				mcCartesianYMoveAbsolute.Execute	:= FALSE;
					IF NOT mcCartesianZMoveAbsolute.Busy THEN
						mcCartesianZMoveAbsolute.Position	:= 380.0;
						mcCartesianZMoveAbsolute.Execute	:= TRUE;	
						iRejectCase		:= 40;
					END_IF
			ELSIF ABS(CartesianYAxisRef.NcToPlc.ActPos - mcCartesianYMoveAbsolute.Position) <= 50.0 THEN	
					bCapCatcher1					:=FALSE;
					bCapCatcher2					:=FALSE;
					bCapCatcher3					:=FALSE;
					bCapCatcher4					:=FALSE;
			END_IF
			
		40:
			IF ABS(CartesianZAxisRef.NcToPlc.ActPos - mcCartesianZMoveAbsolute.Position) <= stParameters.lrBendingDistance AND NOT bCapsBlowON THEN
				bCapsBlowON						:= TRUE;
				bCapBlow1						:= TRUE;
            	bCapBlow2						:= TRUE;
            	bCapBlow3						:= TRUE;
            	bCapBlow4						:= TRUE;
				mcCartesianZMoveAbsolute.Execute	:= FALSE;	
				iRejectCase		:= 50;
			END_IF
	
		50:
			mcCartesianZMoveAbsolute2.Position		:= stParameters.lrTopZPosition;
			mcCartesianZMoveAbsolute2.Acceleration	:= stParameters.lrPickerAcceleration;
			mcCartesianZMoveAbsolute2.Deceleration	:= stParameters.lrPickerAcceleration;
			mcCartesianZMoveAbsolute2.Velocity		:= stParameters.lrPickerSpeed;
			mcCartesianZMoveAbsolute2.Execute		:= TRUE;
				
			mcCartesianYMoveAbsolute.Position	:= stParameters.lrPickYPosition;
			mcCartesianYMoveAbsolute.Execute	:= ABS(CartesianZAxisRef.NcToPlc.ActPos - mcCartesianZMoveAbsolute2.Position) <= stParameters.lrBendingDistance;
			
				IF mcCartesianYMoveAbsolute.Busy THEN
					mcCartesianZMoveAbsolute2.Execute		:= FALSE;
					iRejectCase		:= 60;
				END_IF
				
		60:
			IF 	mcCartesianYMoveAbsolute.Done THEN
				mcCartesianYMoveAbsolute.Execute	:= FALSE;
				bRejectDone							:= TRUE;
			END_IF
	
END_CASE
END_ACTION

ACTION ResetCommands:
	iAbortingCASE									:=0;
	iStoppingCase 									:=0;
	iHomingCase										:=0;
	iErrorResseting2								:=0;
	iTestResetting									:=0;
	iCountAborting									:=0;
	iSimulationCase									:=0;
	diManualModeCase								:=0;

	bEnableLift										:= FALSE;
	mcCartesianYManualMove.JogBackwards				:= FALSE;
	mcCartesianZManualMove.JogBackwards				:= FALSE;
	mcPreScrewerManualMove.JogBackwards				:= FALSE;
	mcCatcherManualMove.JogBackwards				:= FALSE;
	bReject											:= FALSE;
	bRejectDone										:= FALSE;
	bTubeReject										:= FALSE;
	                                        		   
	mcCartesianYManualMove.JogForward				:= FALSE;
	mcCartesianZManualMove.JogForward				:= FALSE;
	mcPreScrewerManualMove.JogForward				:= FALSE;
	mcCatcherManualMove.JogForward					:= FALSE;
	                                        		   
	mcCartesianYStop.Execute						:= FALSE;
	mcCartesianZStop.Execute						:= FALSE;
	mcPreScrewerStop.Execute						:= FALSE;
	mcCatcherStop.Execute							:= FALSE;
	                                        		
	                                        		
	mcCartesianYMoveAbsolute.Execute				:= FALSE;
	mcCartesianZMoveAbsolute.Execute				:= FALSE;
	mcCartesianZMoveAbsolute2.Execute				:= FALSE;
	mcPreScrewerMoveAbsolute.Execute				:= FALSE;
//	mcPreScrewerMoveRelative.Execute				:= FALSE;
	mcCatcherMoveAbsolute.Execute					:= FALSE;
	
	
	fbCartesianYHardReset.Execute					:= FALSE;
	fbCartesianZHardReset.Execute					:= FALSE;
	fbPreScrewerHardReset.Execute					:= FALSE;
	fbCatcherHardReset.Execute						:= FALSE;
	mcCartesianYSoftReset.Execute					:= FALSE;
	mcCartesianZSoftReset.Execute					:= FALSE;
	mcPreScrewerSoftReset.Execute					:= FALSE;
	mcPreScrewerStop.Execute						:= FALSE;
	mcCatcherSoftReset.Execute						:= FALSE;
	mcPreScrewerMoveRelative.Execute				:= FALSE;
	                                        		
	tonVacuumWatchdog.IN							:= FALSE;
//	bMissingCaps									:= FALSE;	
	                                        		
	//bManualCapSucker1								:= FALSE;
	//bManualCapSucker2								:= FALSE;
	//bManualCapSucker3								:= FALSE;
	//bManualCapSucker4								:= FALSE;
	                      	    		    		
	bManualCapBlower1								:= FALSE;
	bManualCapBlower2								:= FALSE;
	bManualCapBlower3								:= FALSE;
	bManualCapBlower4								:= FALSE;
	                       		    	    		
	//bManualCapCatcher1								:= FALSE;
	//bManualCapCatcher2								:= FALSE;
	//bManualCapCatcher3								:= FALSE;
	//bManualCapCatcher4					    		:= FALSE;
	                                        		
	bManualStrawCatchersOpen						:= FALSE;
	bManualStrawCatchersClose						:= FALSE;
	                 			            		
	bManualStrawCatcherActuatorOut					:= FALSE;
	bManualStrawCatcherActuatorIn					:= FALSE; 
	GVL_VIS.bCapSorterPreScrewerBottleCatcherCatch	:= FALSE;
	bAdditionalBlow									:= FALSE;
	bBottleCatcherCatchTemp							:= FALSE;
	
	tonWaitInPlacePos.IN							:= FALSE;
	fbGearInAxisZ.Enable							:= FALSE;
	fbGearInCatcherAxis.Enable						:= FALSE;
	bVirtualMove									:= FALSE;

//	mcCatcherHalt.Execute							:= FALSE;	
//	fbCamTableSelectAxisZ.Execute					:= FALSE;
//	fbCamInAxisZ.Execute							:= FALSE;
//	fbCamTableSelectCatcher.Execute					:= FALSE;
//	fbCamInAxisCatcher.Execute						:= FALSE;
//	fbCamOutAxisCatcher.Execute						:= FALSE;
//	fbCamOutAxisZ.Execute							:= FALSE;
	
(*
iCloseGripperBeforeScrewingCASE		:= 0;
iScrewingCase						:= 0;
iScrewing2Case						:= 0;
iStoppingCase 						:= 0;
iPreparingToReadyCase				:= 0;
iHomingCase							:= 0;
iMStep								:= 0;

iErrorResseting2					:= 0;
iErrorResseting3					:= 0;

mcHeight1GearInMultiMaster.Enable	:=	FALSE;
mcHeight1GearOut.Execute			:=	FALSE;
mcHeight1MoveAbsolute.Execute		:=	FALSE;
mcHeight1MoveAbsolute2.Execute		:=	FALSE;
mcHeight1Stop.Execute				:=	FALSE;
mcHeight1ManualMove.JogBackwards	:=	FALSE;
mcHeight1ManualMove.JogForward		:=	FALSE;
mcHeight1SoftReset					(Execute:=FALSE,Axis:=Height1AxisRef);
fbHeight1HardReset					(Execute:=FALSE,Axis:=Height1AxisRef);

mcHeight2GearInMultiMaster.Enable	:=	FALSE;
mcHeight2GearOut.Execute			:=	FALSE;
mcHeight2MoveAbsolute.Execute		:=	FALSE;
mcHeight2MoveAbsolute2.Execute		:=	FALSE;
mcHeight2Stop.Execute				:=	FALSE;
mcHeight2ManualMove.JogBackwards	:=	FALSE;
mcHeight2ManualMove.JogForward		:=	FALSE;
mcHeight2SoftReset					(Execute:=FALSE,Axis:=Height2AxisRef);
fbHeight2HardReset					(Execute:=FALSE,Axis:=Height2AxisRef);

mcWidthMoveAbsolute.Execute			:=	FALSE;
mcWidthStop.Execute					:=	FALSE;
mcWidthManualMove.JogBackwards		:=	FALSE;
mcWidthManualMove.JogForward		:=	FALSE;
mcWidthSoftReset					(Execute:=FALSE,Axis:=Height2AxisRef);
fbWidthHardReset					(Execute:=FALSE,Axis:=Height2AxisRef);

mcMoveAbsolute.Execute				:=	FALSE;			
mcScrewer1MoveAbsolute.Execute		:=	FALSE;
mcScrewer2MoveAbsolute.Execute		:=	FALSE;
mcScrewer1Stop.Execute				:=	FALSE;
mcScrewer2Stop.Execute				:=	FALSE;
mcScrewer1ManualMove.JogBackwards	:=	FALSE;
mcScrewer1ManualMove.JogForward		:=	FALSE;
mcScrewer2ManualMove.JogBackwards	:=	FALSE;
mcScrewer2ManualMove.JogForward		:=	FALSE;
mcScrewer1MoveVelocity.Execute		:=	FALSE;
mcScrewer2MoveVelocity.Execute		:=	FALSE;
mcScrewer1MoveVelocity2.Execute		:=	FALSE;
mcScrewer2MoveVelocity2.Execute		:=	FALSE;
mcScrewer1TorqueControl.Execute		:=	FALSE;
mcScrewer2TorqueControl.Execute		:=	FALSE;


bStepModeMoving						:=	FALSE;
mcScrewer1SoftReset					(Execute:=FALSE,Axis:=Screwing1AxisRef);	
mcScrewer2SoftReset					(Execute:=FALSE,Axis:=Screwing2AxisRef);	
fbScrewer1HardReset					(Execute:=FALSE,Axis:=Screwing1AxisRef);	
fbScrewer2HardReset					(Execute:=FALSE,Axis:=Screwing2AxisRef);	


//bWasPreparePick1					:=	FALSE;
//bWasPreparePick2					:=	FALSE;	
*)
END_ACTION

ACTION Running:

tonVacuumWatchdog(PT	:= stParameters.tTimeVacuumWatchdog);
bStopAllowed	:= eRunningState = E_CapPreScrewer.eReady OR eRunningState = E_CapPreScrewer.eVerticalDownToCatchPos;

//Otwieranie chwytaków
//bBottleCatcherCatchTemp		R= CartesianZAxisRef.NcToPlc.ActPos < stParameters.lrGripperOpenPosition;
GVL_VIS.bCapSorterPreScrewerBottleCatcherCatch	:= bBottleCatcherCatchTemp AND bCapSorterPreScrewerBottleCatcherEnableShow;
	
tonWaitInPlacePos(PT	:= stParameters.tWaitInPlacePos);
//tonWaitInPlacePos(PT 	:= T#200MS);
eLastRunningState	:= eRunningState;

CASE eRunningState OF

//====================================
	
	(*Oczekiwanie na wykonanie pojedynczego cyklu*)
	E_CapPreScrewer.eReady:

		
		IF NOT bCycleDone AND NOT bCycleNotDone THEN  
                                      	
			IF bRun THEN 
				fbVirtualAxis.fAcceleration				:= stParameters.lrPickerAcceleration;	//100_000_000.0;
				fbVirtualAxis.fDeceleration				:= stParameters.lrPickerAcceleration;	//100_000_000.0;
				fbVirtualAxis.fJerk						:= stParameters.lrPickerJerk;// 	1_000_000;//100_000_000_000;  

				iRejectCase					:= 0;
				bRejectDone					:= FALSE;
				bReject						:= FALSE;
				bTubeReject					:= FALSE;
				
				//Przygotuj do cyklu - otwórz chwytaki
				bCapCatcher1				:= FALSE;
				bCapCatcher2				:= FALSE;
				bCapCatcher3				:= FALSE;
				bCapCatcher4				:= FALSE;
	
				//Wyłącz ssawki
				bCapSucker[1]				:= FALSE;
				bCapSucker[2]				:= FALSE;
				bCapSucker[3]				:= FALSE;
				bCapSucker[4]				:= FALSE;
				//Wyłącz odmuchy
				bCapBlower1					:= FALSE;
				bCapBlower2					:= FALSE;
				bCapBlower3					:= FALSE;
				bCapBlower4					:= FALSE;
				bCapsBlowON					:= FALSE;
				//Otwórz chwytaki słomek
				bStrawCatchersOpen			:= TRUE;
				bStrawCatchersClose			:= FALSE;
				//Cofnij chwytaki słomek
				bStrawCatcherActuatorIn		:= TRUE;
				bStrawCatcherActuatorOut	:= FALSE;
				//Podjedź robotem i chwytakiem słomek w górę jak cofnięty chwytak słomek
				IF tonStrawCatcherIn.Q THEN	
										
					mcCartesianZMoveAbsolute.Execute		:= TRUE;		
					mcCartesianZMoveAbsolute.Position		:= stParameters.lrTopZPosition;
					mcCartesianZMoveAbsolute.Acceleration	:= stParameters.lrPickerAcceleration;
					mcCartesianZMoveAbsolute.Deceleration	:= stParameters.lrPickerAcceleration;
					mcCartesianZMoveAbsolute.Velocity		:= stParameters.lrPickerSpeed;
					
					mcCatcherMoveAbsolute.Execute			:= TRUE;		
					mcCatcherMoveAbsolute.Position			:= stParameters.lrCatcherCatchingPosition;
					mcCatcherMoveAbsolute.Acceleration		:= stParameters.lrCatcherAcceleration;
					mcCatcherMoveAbsolute.Deceleration		:= stParameters.lrCatcherAcceleration;
					mcCatcherMoveAbsolute.Velocity			:= stParameters.lrCatcherSpeed;
					
					//Następny krok
					eRunningState						:= E_CapPreScrewer.ePreparingToPick;
					bCycleNotDone						:= TRUE;
					
				END_IF
				//Reset komendy ruchu osi X
				mcCartesianYMoveAbsolute.Execute		:= FALSE;
				
			END_IF
		END_IF
			
	(*Czekam na pozycję Z w górze i ruszam osią poziomą X na pozycję pobierania i czekam na obie pozycje*)
	E_CapPreScrewer.ePreparingToPick:
		IF (CartesianZAxisRef.NcToPlc.ActPos > stParameters.lrTopZPosition - stParameters.lrBendingDistance) OR
			mcCartesianZMoveAbsolute.Done THEN
			//Jedź osią poziomą X na pozycję pick
			mcCartesianYMoveAbsolute.Execute		:= TRUE;
			mcCartesianYMoveAbsolute.Position		:= stParameters.lrPickYPosition;
			mcCartesianYMoveAbsolute.Acceleration	:= stParameters.lrPickerAcceleration;
			mcCartesianYMoveAbsolute.Deceleration	:= stParameters.lrPickerAcceleration;
			mcCartesianYMoveAbsolute.Velocity		:= stParameters.lrPickerSpeed;
			//Nakrętka pobrana z wózka nr.1
			bMover1InPickPos						:= SEL((stParameters.lrPickYPosition-GVL_Recipe.lrCapSorterPreScrewerPickXMover1PositionShow) <= 0.5, FALSE, TRUE);
			
			//Ustaw obracarkę w pozycji
			mcPreScrewerMoveRelative.Distance		:=  -1 * DINT_TO_LREAL((LREAL_TO_DINT(PreScrewerAxisRef.NcToPlc.SetPos)+diPreSCrewerHomePos) MOD 360);
			mcPreScrewerMoveRelative.Execute		:= mcPreScrewerMoveRelative.Distance<>0;
			mcPreScrewerMoveRelative.Acceleration	:= stParameters.lrScrewAcceleration;
			mcPreScrewerMoveRelative.Deceleration	:= stParameters.lrScrewAcceleration;
			mcPreScrewerMoveRelative.Velocity		:= stParameters.lrScrewSpeed;
		END_IF
		//Jak obie pozycje osiągnięte to wysuń chwytak słomek i następny krok
		IF mcCartesianYMoveAbsolute.Done AND mcCartesianZMoveAbsolute.Done AND mcCatcherMoveAbsolute.Done THEN
			IF mcPreScrewerMoveRelative.Done OR mcPreScrewerMoveRelative.Distance =0 THEN
				//Reset komendy ruchu osi
				mcCartesianYMoveAbsolute.Execute		:= FALSE;
				mcCartesianZMoveAbsolute.Execute		:= FALSE;
				mcPreScrewerMoveRelative.Execute		:= FALSE;
				mcCatcherMoveAbsolute.Execute			:= FALSE;
				//Wysuń chwytaki słomek jesli to potrzebuje recepta        
				bStrawCatcherActuatorIn					:= NOT stParameters.bStrawCatcherON;
				bStrawCatcherActuatorOut				:= stParameters.bStrawCatcherON;    
				//Następny krok
				eRunningState							:= E_CapPreScrewer.ePicking;
			END_IF
		END_IF
		
	
	(*Zjeżdzam na osią pionową Z na pozycję chwytania i załączam ssawki*)		
	E_CapPreScrewer.ePicking:
		//Podjedź robotem w górę	
		mcCartesianZMoveAbsolute.Execute			:= TRUE;		
		mcCartesianZMoveAbsolute.Position			:= stParameters.lrPickZPosition;
		mcCartesianZMoveAbsolute.Acceleration		:= stParameters.lrPickerAcceleration;
		mcCartesianZMoveAbsolute.Deceleration		:= stParameters.lrPickerAcceleration;
		mcCartesianZMoveAbsolute.Velocity			:= stParameters.lrPickerSpeed;
		//Czekam na wykonanie ruchu
		IF mcCartesianZMoveAbsolute.Done THEN
			//Reset komendy ruchu osi
			mcCartesianZMoveAbsolute.Execute		:= FALSE;
			
			//Zeruje rejestry oraz załączanie ssawek
			 FOR i:=1 TO 4 DO
				 bCapSucker[i]						:= stParameters.bPickerActiv[i]; 
				 aCapPresence[i] 					:= FALSE;
			 END_FOR
	
			//Następny krok
			eRunningState							:= E_CapPreScrewer.eVacumCheckPart1;
		END_IF
	
	(*Sprawdzam czy zassane i jazda w górę*)	
	E_CapPreScrewer.eVacumCheckPart1:
		
		tonVacuumWatchdog.IN						:= TRUE;
		
		IF tonSuckedOk[1].Q = stParameters.bPickerActiv[1] AND tonSuckedOk[2].Q = stParameters.bPickerActiv[2]
			AND tonSuckedOk[3].Q = stParameters.bPickerActiv[3] AND tonSuckedOk[4].Q = stParameters.bPickerActiv[4] THEN
			tonVacuumWatchdog.IN					:= FALSE;
		
				FOR i:=1 TO 4 DO
					IF stParameters.bPickerActiv[i] AND stParameters.bStrawCatcherON AND NOT stMoverStatus.stSlotStatus[i].bTubePresent THEN
						bReject								:= TRUE;
						bTubeReject							:= TRUE;
						lrAxisZ_RejectOffset				:= 0.0;
					END_IF

					IF bMover1InPlacePos THEN
						diMover1VacuumRetry[i]		:= 0;
					ELSE
						diMover2VacuumRetry[i]		:= 0;
					END_IF	
				END_FOR 
				
			eRunningState 							:= E_CapPreScrewer.eVacumCheckPart2;
	
		ELSIF tonVacuumWatchdog.Q THEN
		
			FOR i:=1 TO 4 DO
				bCapSucker[i]							:= tonSuckedOk[i].Q;
				
				//robimy odrzut jeżeli zostanie wykryto brak słomki
				IF stParameters.bPickerActiv[i] AND stParameters.bStrawCatcherON AND NOT stMoverStatus.stSlotStatus[i].bTubePresent THEN
					bReject								:= TRUE;
					bTubeReject							:= TRUE;
					lrAxisZ_RejectOffset				:= 0.0;
				END_IF
				
						//Detekcja niepobranej nasadki --> odrzut aktywowany opcjonalnie z receptury
					IF stParameters.bPickerActiv[i] AND NOT tonSuckedOk[i].Q AND NOT stParameters.bVacuumDeactivate THEN
						bReject							:= SEL(stParameters.bRejectON, bReject, TRUE);
						lrAxisZ_RejectOffset			:= SEL(stParameters.bRejectON, lrAxisZ_RejectOffset, 13.0);	//offset dodatkowego zjazdu kartezjanem 
						
						IF bMover1InPlacePos THEN
							diMover1VacuumRetry[i]		:= diMover1VacuumRetry[i] + 1;
						ELSE	
							diMover2VacuumRetry[i]		:= diMover2VacuumRetry[i] + 1;
						END_IF
					ELSIF tonSuckedOk[i].Q OR stParameters.bVacuumDeactivate THEN
						IF 	bMover1InPlacePos THEN
							diMover1VacuumRetry[i]		:= 0;
						ELSE
							diMover2VacuumRetry[i]		:= 0;
						END_IF	
					END_IF	
	    	
			END_FOR
				tonVacuumWatchdog.IN					:= FALSE;
				eRunningState 							:= E_CapPreScrewer.eVacumCheckPart2;
	
		END_IF
		
		
	E_CapPreScrewer.eVacumCheckPart2:	
			
		//Jezeli nie jest przyssana zadna nasadka to pdjezdzamy na poz. ready oraz wystawiamy flage bMissingCaps
		IF bReject THEN
			Reject();
				IF bRejectDone THEN				
					eRunningState						:= E_CapPreScrewer.eReady;	
				END_IF		
		ELSIF NOT tonSuckedOk[1].Q AND NOT tonSuckedOk[2].Q AND NOT tonSuckedOk[3].Q AND NOT tonSuckedOk[4].Q THEN
			bCapSucker[1]							:= FALSE;
			bCapSucker[2]							:= False;
			bCapSucker[3]							:= False;
		    bCapSucker[4]							:= False;	
			mcCartesianZMoveAbsolute.Execute		:= TRUE;		
			mcCartesianZMoveAbsolute.Position		:= stParameters.lrTopZPosition;
			mcCartesianZMoveAbsolute.Acceleration	:= stParameters.lrPickerAcceleration;
			mcCartesianZMoveAbsolute.Deceleration	:= stParameters.lrPickerAcceleration;
			mcCartesianZMoveAbsolute.Velocity		:= stParameters.lrPickerSpeed;
			
